LIN {X 0,Y 136.202,Z 770.659,A -85,B 0,C 180,E1 7477.588,E2 7477.588} C_VEL
LIN {X 0,Y 136.38,Z 770.694,A -85,B 0,C 180,E1 7471.676,E2 7471.676} C_VEL
LIN {X 0,Y 136.378,Z 769.624,A -85,B 0,C 180,E1 7466.633,E2 7466.633} C_VEL
LIN {X 0,Y 136.448,Z 766.979,A -85,B 0,C 180,E1 7460.718,E2 7460.718} C_VEL
LIN {X 0,Y 136.634,Z 766.026,A -85,B 0,C 180,E1 7458.6,E2 7458.6} C_VEL
LIN {X 0,Y 138.841,Z 767.204,A -85,B 0,C 180,E1 7448.274,E2 7448.274} C_VEL
LIN {X 0,Y 145.472,Z 766.561,A -85,B 0,C 180,E1 7438.042,E2 7438.042} C_VEL
LIN {X 0,Y 157.729,Z 763.951,A -85,B 0,C 180,E1 7428.267,E2 7428.267} C_VEL
LIN {X 0,Y 170.729,Z 760.685,A -85,B 0,C 180,E1 7421.759,E2 7421.759} C_VEL
LIN {X 0,Y 156.243,Z 761.337,A -85,B 0,C 180,E1 7414.272,E2 7414.272} C_VEL
LIN {X 0,Y 145.762,Z 760.293,A -85,B 0,C 180,E1 7405.603,E2 7405.603} C_VEL
LIN {X 0,Y 139.457,Z 757.48,A -85,B 0,C 180,E1 7396.236,E2 7396.236} C_VEL
LIN {X 0,Y 136.886,Z 753.335,A -85,B 0,C 180,E1 7387.553,E2 7387.553} C_VEL
LIN {X 0,Y 136.308,Z 748.658,A -85,B 0,C 180,E1 7380.419,E2 7380.419} C_VEL
LIN {X 0,Y 136.364,Z 742.798,A -85,B 0,C 180,E1 7373.684,E2 7373.684} C_VEL
LIN {X 0,Y 137.263,Z 734.901,A -85,B 0,C 180,E1 7366.519,E2 7366.519} C_VEL
LIN {X 0,Y 139.461,Z 725.036,A -85,B 0,C 180,E1 7359.431,E2 7359.431} C_VEL
LIN {X 0,Y 142.943,Z 713.689,A -85,B 0,C 180,E1 7352.955,E2 7352.955} C_VEL
LIN {X 0,Y 147.839,Z 700.038,A -85,B 0,C 180,E1 7346.781,E2 7346.781} C_VEL
LIN {X 0,Y 153.697,Z 684.691,A -85,B 0,C 180,E1 7341.325,E2 7341.325} C_VEL
LIN {X 0,Y 160.141,Z 667.742,A -85,B 0,C 180,E1 7336.621,E2 7336.621} C_VEL
LIN {X 0,Y 166.838,Z 649.18,A -85,B 0,C 180,E1 7332.63,E2 7332.63} C_VEL
LIN {X 0,Y 173.319,Z 629.638,A -85,B 0,C 180,E1 7329.371,E2 7329.371} C_VEL
LIN {X 0,Y 179.516,Z 608.54,A -85,B 0,C 180,E1 7326.672,E2 7326.672} C_VEL
LIN {X 0,Y 184.868,Z 587.205,A -85,B 0,C 180,E1 7324.607,E2 7324.607} C_VEL
LIN {X 0,Y 189.518,Z 564.355,A -85,B 0,C 180,E1 7323.014,E2 7323.014} C_VEL
LIN {X 0,Y 200.571,Z 495.538,A -85,B 0,C 180,E1 7319.493,E2 7319.493} C_VEL
LIN {X 0,Y 196.571,Z 500.049,A -85,B 0,C 180,E1 7318.892,E2 7318.892} C_VEL
LIN {X 0,Y 192.978,Z 508.1,A -85,B 0,C 180,E1 7318.713,E2 7318.713} C_VEL
LIN {X 0,Y 189.976,Z 512.133,A -85,B 0,C 180,E1 7318.319,E2 7318.319} C_VEL
LIN {X 0,Y 187.942,Z 514.262,A -85,B 0,C 180,E1 7317.832,E2 7317.832} C_VEL
LIN {X 0,Y 187.389,Z 518.122,A -85,B 0,C 180,E1 7317.404,E2 7317.404} C_VEL
LIN {X 0,Y 186.903,Z 526.414,A -85,B 0,C 180,E1 7317.05,E2 7317.05} C_VEL
LIN {X 0,Y 178.232,Z 635.184,A -85,B 0,C 180,E1 7313.3,E2 7313.3} C_VEL
LIN {X 0,Y 175.765,Z 651.989,A -85,B 0,C 180,E1 7312.165,E2 7312.165} C_VEL
LIN {X 0,Y 172.642,Z 666.742,A -85,B 0,C 180,E1 7310.692,E2 7310.692} C_VEL
LIN {X 0,Y 168.594,Z 681.234,A -85,B 0,C 180,E1 7308.682,E2 7308.682} C_VEL
LIN {X 0,Y 163.629,Z 695.775,A -85,B 0,C 180,E1 7305.964,E2 7305.964} C_VEL
LIN {X 0,Y 158.471,Z 708.511,A -85,B 0,C 180,E1 7302.762,E2 7302.762} C_VEL
LIN {X 0,Y 153.349,Z 719.856,A -85,B 0,C 180,E1 7299.007,E2 7299.007} C_VEL
LIN {X 0,Y 148.442,Z 729.85,A -85,B 0,C 180,E1 7294.64,E2 7294.64} C_VEL
LIN {X 0,Y 143.727,Z 739.095,A -85,B 0,C 180,E1 7289.207,E2 7289.207} C_VEL
LIN {X 0,Y 140.182,Z 746.209,A -85,B 0,C 180,E1 7283.452,E2 7283.452} C_VEL
LIN {X 0,Y 137.716,Z 751.82,A -85,B 0,C 180,E1 7276.998,E2 7276.998} C_VEL
LIN {X 0,Y 136.594,Z 755.376,A -85,B 0,C 180,E1 7270.773,E2 7270.773} C_VEL
LIN {X 0,Y 136.355,Z 757.366,A -85,B 0,C 180,E1 7264.371,E2 7264.371} C_VEL
LIN {X 0,Y 136.925,Z 757.835,A -85,B 0,C 180,E1 7257.793,E2 7257.793} C_VEL
LIN {X 0,Y 138.691,Z 756.654,A -85,B 0,C 180,E1 7251.135,E2 7251.135} C_VEL
LIN {X 0,Y 142.253,Z 753.429,A -85,B 0,C 180,E1 7244.205,E2 7244.205} C_VEL
LIN {X 0,Y 147.052,Z 748.647,A -85,B 0,C 180,E1 7238.226,E2 7238.226} C_VEL
LIN {X 0,Y 153.218,Z 741.888,A -85,B 0,C 180,E1 7232.676,E2 7232.676} C_VEL
LIN {X 0,Y 160.059,Z 733.612,A -85,B 0,C 180,E1 7227.939,E2 7227.939} C_VEL
LIN {X 0,Y 167.558,Z 723.336,A -85,B 0,C 180,E1 7223.747,E2 7223.747} C_VEL
LIN {X 0,Y 174.867,Z 711.855,A -85,B 0,C 180,E1 7220.34,E2 7220.34} C_VEL
LIN {X 0,Y 181.888,Z 698.953,A -85,B 0,C 180,E1 7217.509,E2 7217.509} C_VEL
LIN {X 0,Y 188.022,Z 685.344,A -85,B 0,C 180,E1 7215.305,E2 7215.305} C_VEL
LIN {X 0,Y 193.337,Z 670.636,A -85,B 0,C 180,E1 7213.545,E2 7213.545} C_VEL
LIN {X 0,Y 197.488,Z 655.424,A -85,B 0,C 180,E1 7212.23,E2 7212.23} C_VEL
LIN {X 0,Y 200.617,Z 638.603,A -85,B 0,C 180,E1 7211.246,E2 7211.246} C_VEL
LIN {X 0,Y 204.02,Z 605.103,A -85,B 0,C 180,E1 7210.152,E2 7210.152} C_VEL
LIN {X 0,Y 211.834,Z 524.075,A -85,B 0,C 180,E1 7207.779,E2 7207.779} C_VEL
LIN {X 0,Y 212.398,Z 496.448,A -85,B 0,C 180,E1 7205.573,E2 7205.573} C_VEL
LIN {X 0,Y 212.772,Z 490.461,A -85,B 0,C 180,E1 7205.02,E2 7205.02} C_VEL
LIN {X 0,Y 224.955,Z 447.879,A -85,B 0,C 180,E1 7199.89,E2 7199.89} C_VEL
LIN {X 0,Y 225.289,Z 446.689,A -85,B 0,C 180,E1 7199.747,E2 7199.747} C_VEL
LIN {X 0,Y 224.925,Z 439.714,A -85,B 0,C 180,E1 7196.433,E2 7196.433} C_VEL
LIN {X 0,Y 224.669,Z 434.477,A -85,B 0,C 180,E1 7192.917,E2 7192.917} C_VEL
LIN {X 0,Y 224.564,Z 431.171,A -85,B 0,C 180,E1 7189.714,E2 7189.714} C_VEL
LIN {X 0,Y 225.058,Z 428.722,A -85,B 0,C 180,E1 7185.858,E2 7185.858} C_VEL
LIN {X 0,Y 225.213,Z 428.615,A -85,B 0,C 180,E1 7184.024,E2 7184.024} C_VEL
LIN {X 0,Y 223.089,Z 438.023,A -85,B 0,C 180,E1 7180.503,E2 7180.503} C_VEL
LIN {X 0,Y 222.438,Z 440.67,A -85,B 0,C 180,E1 7179.938,E2 7179.938} C_VEL
LIN {X 0,Y 221.128,Z 444.689,A -85,B 0,C 180,E1 7179.659,E2 7179.659} C_VEL
LIN {X 0,Y 216.142,Z 458.259,A -85,B 0,C 180,E1 7179.808,E2 7179.808} C_VEL
LIN {X 0,Y 215.382,Z 460.548,A -85,B 0,C 180,E1 7179.71,E2 7179.71} C_VEL
LIN {X 0,Y 204.017,Z 497.28,A -85,B 0,C 180,E1 7177.4,E2 7177.4} C_VEL
LIN {X 0,Y 194.372,Z 587.356,A -85,B 0,C 180,E1 7174.197,E2 7174.197} C_VEL
LIN {X 0,Y 190.852,Z 624.419,A -85,B 0,C 180,E1 7172.598,E2 7172.598} C_VEL
LIN {X 0,Y 188.404,Z 647.642,A -85,B 0,C 180,E1 7171.449,E2 7171.449} C_VEL
LIN {X 0,Y 185.307,Z 663.835,A -85,B 0,C 180,E1 7170.239,E2 7170.239} C_VEL
LIN {X 0,Y 180.934,Z 679.336,A -85,B 0,C 180,E1 7168.617,E2 7168.617} C_VEL
LIN {X 0,Y 175.515,Z 694.069,A -85,B 0,C 180,E1 7166.563,E2 7166.563} C_VEL
LIN {X 0,Y 169.269,Z 707.769,A -85,B 0,C 180,E1 7164.015,E2 7164.015} C_VEL
LIN {X 0,Y 161.79,Z 721.666,A -85,B 0,C 180,E1 7160.572,E2 7160.572} C_VEL
LIN {X 0,Y 154.309,Z 733.62,A -85,B 0,C 180,E1 7156.522,E2 7156.522} C_VEL
LIN {X 0,Y 147.122,Z 744.014,A -85,B 0,C 180,E1 7151.754,E2 7151.754} C_VEL
LIN {X 0,Y 140.559,Z 752.753,A -85,B 0,C 180,E1 7146.181,E2 7146.181} C_VEL
LIN {X 0,Y 135.035,Z 759.962,A -85,B 0,C 180,E1 7139.736,E2 7139.736} C_VEL
LIN {X 0,Y 131.03,Z 765.309,A -85,B 0,C 180,E1 7132.586,E2 7132.586} C_VEL
LIN {X 0,Y 128.834,Z 768.723,A -85,B 0,C 180,E1 7125.294,E2 7125.294} C_VEL
LIN {X 0,Y 128.211,Z 770.292,A -85,B 0,C 180,E1 7117.951,E2 7117.951} C_VEL
LIN {X 0,Y 128.388,Z 770.241,A -85,B 0,C 180,E1 7111.78,E2 7111.78} C_VEL
LIN {X 0,Y 128.386,Z 769.096,A -85,B 0,C 180,E1 7106.423,E2 7106.423} C_VEL
LIN {X 0,Y 128.497,Z 766.359,A -85,B 0,C 180,E1 7100.138,E2 7100.138} C_VEL
LIN {X 0,Y 128.816,Z 764.854,A -85,B 0,C 180,E1 7097.443,E2 7097.443} C_VEL
LIN {X 0,Y 131.253,Z 766.254,A -85,B 0,C 180,E1 7087.134,E2 7087.134} C_VEL
LIN {X 0,Y 138.611,Z 765.981,A -85,B 0,C 180,E1 7076.255,E2 7076.255} C_VEL
LIN {X 0,Y 152.308,Z 763.787,A -85,B 0,C 180,E1 7065.899,E2 7065.899} C_VEL
LIN {X 0,Y 160.499,Z 762.17,A -85,B 0,C 180,E1 7061.711,E2 7061.711} C_VEL
LIN {X 0,Y 146.19,Z 761.822,A -85,B 0,C 180,E1 7053.64,E2 7053.64} C_VEL
LIN {X 0,Y 136.487,Z 759.886,A -85,B 0,C 180,E1 7044.679,E2 7044.679} C_VEL
LIN {X 0,Y 130.847,Z 756.352,A -85,B 0,C 180,E1 7035.057,E2 7035.057} C_VEL
LIN {X 0,Y 128.672,Z 751.44,A -85,B 0,C 180,E1 7025.796,E2 7025.796} C_VEL
LIN {X 0,Y 128.309,Z 746.391,A -85,B 0,C 180,E1 7018.659,E2 7018.659} C_VEL
LIN {X 0,Y 128.557,Z 739.855,A -85,B 0,C 180,E1 7011.5,E2 7011.5} C_VEL
LIN {X 0,Y 129.878,Z 731.149,A -85,B 0,C 180,E1 7003.908,E2 7003.908} C_VEL
LIN {X 0,Y 132.724,Z 720.359,A -85,B 0,C 180,E1 6996.466,E2 6996.466} C_VEL
LIN {X 0,Y 136.933,Z 708.027,A -85,B 0,C 180,E1 6989.745,E2 6989.745} C_VEL
LIN {X 0,Y 142.425,Z 693.704,A -85,B 0,C 180,E1 6983.613,E2 6983.613} C_VEL
LIN {X 0,Y 148.518,Z 678.345,A -85,B 0,C 180,E1 6978.459,E2 6978.459} C_VEL
LIN {X 0,Y 155.327,Z 660.805,A -85,B 0,C 180,E1 6973.864,E2 6973.864} C_VEL
LIN {X 0,Y 162.096,Z 642.235,A -85,B 0,C 180,E1 6970.102,E2 6970.102} C_VEL
LIN {X 0,Y 168.842,Z 621.674,A -85,B 0,C 180,E1 6966.92,E2 6966.92} C_VEL
LIN {X 0,Y 175.053,Z 600.001,A -85,B 0,C 180,E1 6964.374,E2 6964.374} C_VEL
LIN {X 0,Y 180.378,Z 577.861,A -85,B 0,C 180,E1 6962.439,E2 6962.439} C_VEL
LIN {X 0,Y 184.961,Z 553.44,A -85,B 0,C 180,E1 6960.942,E2 6960.942} C_VEL
LIN {X 0,Y 189.625,Z 524.883,A -85,B 0,C 180,E1 6959.422,E2 6959.422} C_VEL
LIN {X 0,Y 185.421,Z 534.382,A -85,B 0,C 180,E1 6959.255,E2 6959.255} C_VEL
LIN {X 0,Y 182.143,Z 538.992,A -85,B 0,C 180,E1 6958.845,E2 6958.845} C_VEL
LIN {X 0,Y 180.549,Z 542.085,A -85,B 0,C 180,E1 6958.47,E2 6958.47} C_VEL
LIN {X 0,Y 179.354,Z 551.32,A -85,B 0,C 180,E1 6958.045,E2 6958.045} C_VEL
LIN {X 0,Y 172.354,Z 635.636,A -85,B 0,C 180,E1 6955.07,E2 6955.07} C_VEL
LIN {X 0,Y 169.761,Z 652.518,A -85,B 0,C 180,E1 6953.913,E2 6953.913} C_VEL
LIN {X 0,Y 166.535,Z 667.111,A -85,B 0,C 180,E1 6952.433,E2 6952.433} C_VEL
LIN {X 0,Y 162.279,Z 681.697,A -85,B 0,C 180,E1 6950.376,E2 6950.376} C_VEL
LIN {X 0,Y 157.086,Z 696.228,A -85,B 0,C 180,E1 6947.602,E2 6947.602} C_VEL
LIN {X 0,Y 151.421,Z 709.519,A -85,B 0,C 180,E1 6944.146,E2 6944.146} C_VEL
LIN {X 0,Y 146.063,Z 720.768,A -85,B 0,C 180,E1 6940.256,E2 6940.256} C_VEL
LIN {X 0,Y 140.524,Z 731.368,A -85,B 0,C 180,E1 6935.312,E2 6935.312} C_VEL
LIN {X 0,Y 135.971,Z 739.819,A -85,B 0,C 180,E1 6930.005,E2 6930.005} C_VEL
LIN {X 0,Y 132.256,Z 746.841,A -85,B 0,C 180,E1 6923.929,E2 6923.929} C_VEL
LIN {X 0,Y 129.696,Z 752.395,A -85,B 0,C 180,E1 6917.086,E2 6917.086} C_VEL
LIN {X 0,Y 128.544,Z 755.948,A -85,B 0,C 180,E1 6910.256,E2 6910.256} C_VEL
LIN {X 0,Y 128.396,Z 757.896,A -85,B 0,C 180,E1 6903.155,E2 6903.155} C_VEL
LIN {X 0,Y 129.213,Z 758.215,A -85,B 0,C 180,E1 6896.148,E2 6896.148} C_VEL
LIN {X 0,Y 131.554,Z 756.704,A -85,B 0,C 180,E1 6888.804,E2 6888.804} C_VEL
LIN {X 0,Y 135.603,Z 753.414,A -85,B 0,C 180,E1 6881.873,E2 6881.873} C_VEL
LIN {X 0,Y 141.262,Z 748.146,A -85,B 0,C 180,E1 6875.481,E2 6875.481} C_VEL
LIN {X 0,Y 147.897,Z 741.367,A -85,B 0,C 180,E1 6870.02,E2 6870.02} C_VEL
LIN {X 0,Y 155.646,Z 732.426,A -85,B 0,C 180,E1 6865.084,E2 6865.084} C_VEL
LIN {X 0,Y 163.193,Z 722.607,A -85,B 0,C 180,E1 6861.193,E2 6861.193} C_VEL
LIN {X 0,Y 170.7,Z 711.251,A -85,B 0,C 180,E1 6857.926,E2 6857.926} C_VEL
LIN {X 0,Y 177.733,Z 698.817,A -85,B 0,C 180,E1 6855.265,E2 6855.265} C_VEL
LIN {X 0,Y 184.25,Z 684.766,A -85,B 0,C 180,E1 6853.06,E2 6853.06} C_VEL
LIN {X 0,Y 189.682,Z 670.139,A -85,B 0,C 180,E1 6851.368,E2 6851.368} C_VEL
LIN {X 0,Y 194.005,Z 654.43,A -85,B 0,C 180,E1 6850.073,E2 6850.073} C_VEL
LIN {X 0,Y 197.094,Z 637.969,A -85,B 0,C 180,E1 6849.154,E2 6849.154} C_VEL
LIN {X 0,Y 208.623,Z 525.21,A -85,B 0,C 180,E1 6845.796,E2 6845.796} C_VEL
LIN {X 0,Y 209.509,Z 497.097,A -85,B 0,C 180,E1 6843.507,E2 6843.507} C_VEL
LIN {X 0,Y 209.986,Z 490.835,A -85,B 0,C 180,E1 6842.913,E2 6842.913} C_VEL
LIN {X 0,Y 221.687,Z 451.523,A -85,B 0,C 180,E1 6838.224,E2 6838.224} C_VEL
LIN {X 0,Y 221.644,Z 445.832,A -85,B 0,C 180,E1 6835.343,E2 6835.343} C_VEL
LIN {X 0,Y 221.626,Z 441.035,A -85,B 0,C 180,E1 6831.961,E2 6831.961} C_VEL
LIN {X 0,Y 221.723,Z 438.353,A -85,B 0,C 180,E1 6829.083,E2 6829.083} C_VEL
LIN {X 0,Y 222.268,Z 436.205,A -85,B 0,C 180,E1 6825.676,E2 6825.676} C_VEL
LIN {X 0,Y 222.344,Z 436.178,A -85,B 0,C 180,E1 6824.615,E2 6824.615} C_VEL
LIN {X 0,Y 219.694,Z 447.341,A -85,B 0,C 180,E1 6820.491,E2 6820.491} C_VEL
LIN {X 0,Y 215.382,Z 460.548,A -85,B 0,C 180,E1 6819.71,E2 6819.71} C_VEL
LIN {X 0,Y 212.886,Z 467.853,A -85,B 0,C 180,E1 6819.514,E2 6819.514} C_VEL
LIN {X 0,Y 205.414,Z 487.684,A -85,B 0,C 180,E1 6820.021,E2 6820.021} C_VEL
LIN {X 0,Y 203.249,Z 493.872,A -85,B 0,C 180,E1 6819.814,E2 6819.814} C_VEL
LIN {X 0,Y 202.069,Z 500.702,A -85,B 0,C 180,E1 6819.5,E2 6819.5} C_VEL
LIN {X 0,Y 192.265,Z 588.417,A -85,B 0,C 180,E1 6816.467,E2 6816.467} C_VEL
LIN {X 0,Y 188.432,Z 625.593,A -85,B 0,C 180,E1 6814.875,E2 6814.875} C_VEL
LIN {X 0,Y 185.928,Z 647.063,A -85,B 0,C 180,E1 6813.826,E2 6813.826} C_VEL
LIN {X 0,Y 182.619,Z 663.38,A -85,B 0,C 180,E1 6812.656,E2 6812.656} C_VEL
LIN {X 0,Y 178.11,Z 678.587,A -85,B 0,C 180,E1 6811.124,E2 6811.124} C_VEL
LIN {X 0,Y 172.036,Z 694.227,A -85,B 0,C 180,E1 6809.002,E2 6809.002} C_VEL
LIN {X 0,Y 165.087,Z 708.426,A -85,B 0,C 180,E1 6806.377,E2 6806.377} C_VEL
LIN {X 0,Y 157.471,Z 721.539,A -85,B 0,C 180,E1 6803.126,E2 6803.126} C_VEL
LIN {X 0,Y 149.139,Z 733.82,A -85,B 0,C 180,E1 6798.929,E2 6798.929} C_VEL
LIN {X 0,Y 141.683,Z 743.714,A -85,B 0,C 180,E1 6794.311,E2 6794.311} C_VEL
LIN {X 0,Y 134.485,Z 752.399,A -85,B 0,C 180,E1 6788.64,E2 6788.64} C_VEL
LIN {X 0,Y 128.322,Z 759.579,A -85,B 0,C 180,E1 6781.989,E2 6781.989} C_VEL
LIN {X 0,Y 123.87,Z 764.727,A -85,B 0,C 180,E1 6774.812,E2 6774.812} C_VEL
LIN {X 0,Y 121.103,Z 768.31,A -85,B 0,C 180,E1 6766.791,E2 6766.791} C_VEL
LIN {X 0,Y 120.228,Z 769.872,A -85,B 0,C 180,E1 6759.086,E2 6759.086} C_VEL
LIN {X 0,Y 120.376,Z 769.844,A -85,B 0,C 180,E1 6752.375,E2 6752.375} C_VEL
LIN {X 0,Y 120.409,Z 768.863,A -85,B 0,C 180,E1 6747.139,E2 6747.139} C_VEL
LIN {X 0,Y 120.475,Z 766.241,A -85,B 0,C 180,E1 6740.44,E2 6740.44} C_VEL
LIN {X 0,Y 121.104,Z 763.691,A -85,B 0,C 180,E1 6735.654,E2 6735.654} C_VEL
LIN {X 0,Y 124.727,Z 765.297,A -85,B 0,C 180,E1 6723.833,E2 6723.833} C_VEL
LIN {X 0,Y 134.486,Z 765.11,A -85,B 0,C 180,E1 6711.892,E2 6711.892} C_VEL
LIN {X 0,Y 149.618,Z 763.223,A -85,B 0,C 180,E1 6702.111,E2 6702.111} C_VEL
LIN {X 0,Y 150.332,Z 763.087,A -85,B 0,C 180,E1 6701.688,E2 6701.688} C_VEL
LIN {X 0,Y 136.634,Z 761.817,A -85,B 0,C 180,E1 6693.285,E2 6693.285} C_VEL
LIN {X 0,Y 126.957,Z 758.851,A -85,B 0,C 180,E1 6683.188,E2 6683.188} C_VEL
LIN {X 0,Y 122.02,Z 754.358,A -85,B 0,C 180,E1 6672.78,E2 6672.78} C_VEL
LIN {X 0,Y 120.548,Z 749.125,A -85,B 0,C 180,E1 6663.803,E2 6663.803} C_VEL
LIN {X 0,Y 120.361,Z 743.74,A -85,B 0,C 180,E1 6656.665,E2 6656.665} C_VEL
LIN {X 0,Y 120.871,Z 736.504,A -85,B 0,C 180,E1 6649.03,E2 6649.03} C_VEL
LIN {X 0,Y 122.746,Z 726.938,A -85,B 0,C 180,E1 6640.982,E2 6640.982} C_VEL
LIN {X 0,Y 126.078,Z 715.923,A -85,B 0,C 180,E1 6633.632,E2 6633.632} C_VEL
LIN {X 0,Y 130.65,Z 703.573,A -85,B 0,C 180,E1 6627.085,E2 6627.085} C_VEL
LIN {X 0,Y 136.581,Z 688.898,A -85,B 0,C 180,E1 6620.979,E2 6620.979} C_VEL
LIN {X 0,Y 143.505,Z 671.986,A -85,B 0,C 180,E1 6615.553,E2 6615.553} C_VEL
LIN {X 0,Y 150.649,Z 653.881,A -85,B 0,C 180,E1 6611.081,E2 6611.081} C_VEL
LIN {X 0,Y 157.86,Z 634.093,A -85,B 0,C 180,E1 6607.352,E2 6607.352} C_VEL
LIN {X 0,Y 164.696,Z 612.92,A -85,B 0,C 180,E1 6604.343,E2 6604.343} C_VEL
LIN {X 0,Y 170.893,Z 590.458,A -85,B 0,C 180,E1 6601.963,E2 6601.963} C_VEL
LIN {X 0,Y 176.109,Z 567.407,A -85,B 0,C 180,E1 6600.197,E2 6600.197} C_VEL
LIN {X 0,Y 176.373,Z 565.822,A -85,B 0,C 180,E1 6600.091,E2 6600.091} C_VEL
LIN {X 0,Y 173.022,Z 569.857,A -85,B 0,C 180,E1 6599.518,E2 6599.518} C_VEL
LIN {X 0,Y 171.94,Z 575.214,A -85,B 0,C 180,E1 6599.172,E2 6599.172} C_VEL
LIN {X 0,Y 166.523,Z 636.559,A -85,B 0,C 180,E1 6596.913,E2 6596.913} C_VEL
LIN {X 0,Y 163.719,Z 653.78,A -85,B 0,C 180,E1 6595.701,E2 6595.701} C_VEL
LIN {X 0,Y 160.202,Z 668.669,A -85,B 0,C 180,E1 6594.133,E2 6594.133} C_VEL
LIN {X 0,Y 155.492,Z 683.807,A -85,B 0,C 180,E1 6591.902,E2 6591.902} C_VEL
LIN {X 0,Y 150.342,Z 697.358,A -85,B 0,C 180,E1 6589.195,E2 6589.195} C_VEL
LIN {X 0,Y 144.245,Z 710.887,A -85,B 0,C 180,E1 6585.522,E2 6585.522} C_VEL
LIN {X 0,Y 138.832,Z 721.611,A -85,B 0,C 180,E1 6581.624,E2 6581.624} C_VEL
LIN {X 0,Y 133.031,Z 732.092,A -85,B 0,C 180,E1 6576.478,E2 6576.478} C_VEL
LIN {X 0,Y 128.241,Z 740.48,A -85,B 0,C 180,E1 6570.898,E2 6570.898} C_VEL
LIN {X 0,Y 124.337,Z 747.428,A -85,B 0,C 180,E1 6564.468,E2 6564.468} C_VEL
LIN {X 0,Y 121.672,Z 752.937,A -85,B 0,C 180,E1 6557.186,E2 6557.186} C_VEL
LIN {X 0,Y 120.494,Z 756.527,A -85,B 0,C 180,E1 6549.609,E2 6549.609} C_VEL
LIN {X 0,Y 120.441,Z 758.339,A -85,B 0,C 180,E1 6542.303,E2 6542.303} C_VEL
LIN {X 0,Y 121.474,Z 758.594,A -85,B 0,C 180,E1 6534.825,E2 6534.825} C_VEL
LIN {X 0,Y 124.311,Z 756.97,A -85,B 0,C 180,E1 6526.876,E2 6526.876} C_VEL
LIN {X 0,Y 128.808,Z 753.656,A -85,B 0,C 180,E1 6519.791,E2 6519.791} C_VEL
LIN {X 0,Y 135.028,Z 748.367,A -85,B 0,C 180,E1 6513.212,E2 6513.212} C_VEL
LIN {X 0,Y 142.225,Z 741.57,A -85,B 0,C 180,E1 6507.646,E2 6507.646} C_VEL
LIN {X 0,Y 149.895,Z 733.32,A -85,B 0,C 180,E1 6503.011,E2 6503.011} C_VEL
LIN {X 0,Y 158.003,Z 723.418,A -85,B 0,C 180,E1 6499.025,E2 6499.025} C_VEL
LIN {X 0,Y 165.979,Z 712.006,A -85,B 0,C 180,E1 6495.73,E2 6495.73} C_VEL
LIN {X 0,Y 173.692,Z 698.979,A -85,B 0,C 180,E1 6492.975,E2 6492.975} C_VEL
LIN {X 0,Y 180.303,Z 685.283,A -85,B 0,C 180,E1 6490.869,E2 6490.869} C_VEL
LIN {X 0,Y 186.029,Z 670.575,A -85,B 0,C 180,E1 6489.195,E2 6489.195} C_VEL
LIN {X 0,Y 190.559,Z 654.845,A -85,B 0,C 180,E1 6487.92,E2 6487.92} C_VEL
LIN {X 0,Y 193.788,Z 638.429,A -85,B 0,C 180,E1 6487.022,E2 6487.022} C_VEL
LIN {X 0,Y 204.252,Z 540.88,A -85,B 0,C 180,E1 6484.199,E2 6484.199} C_VEL
LIN {X 0,Y 205.73,Z 526.209,A -85,B 0,C 180,E1 6483.739,E2 6483.739} C_VEL
LIN {X 0,Y 206.965,Z 497.506,A -85,B 0,C 180,E1 6481.357,E2 6481.357} C_VEL
LIN {X 0,Y 207.351,Z 491.943,A -85,B 0,C 180,E1 6480.83,E2 6480.83} C_VEL
LIN {X 0,Y 218.321,Z 456.356,A -85,B 0,C 180,E1 6476.621,E2 6476.621} C_VEL
LIN {X 0,Y 218.508,Z 451.219,A -85,B 0,C 180,E1 6473.696,E2 6473.696} C_VEL
LIN {X 0,Y 218.611,Z 447.258,A -85,B 0,C 180,E1 6470.524,E2 6470.524} C_VEL
LIN {X 0,Y 218.922,Z 445.339,A -85,B 0,C 180,E1 6468.141,E2 6468.141} C_VEL
LIN {X 0,Y 219.533,Z 443.702,A -85,B 0,C 180,E1 6465.258,E2 6465.258} C_VEL
LIN {X 0,Y 217.397,Z 451.382,A -85,B 0,C 180,E1 6462.388,E2 6462.388} C_VEL
LIN {X 0,Y 203.249,Z 493.872,A -85,B 0,C 180,E1 6459.814,E2 6459.814} C_VEL
LIN {X 0,Y 202.26,Z 498.075,A -85,B 0,C 180,E1 6459.759,E2 6459.759} C_VEL
LIN {X 0,Y 198.78,Z 519.875,A -85,B 0,C 180,E1 6460.87,E2 6460.87} C_VEL
LIN {X 0,Y 197.506,Z 528.802,A -85,B 0,C 180,E1 6460.868,E2 6460.868} C_VEL
LIN {X 0,Y 190.628,Z 588.142,A -85,B 0,C 180,E1 6458.825,E2 6458.825} C_VEL
LIN {X 0,Y 186.453,Z 626.377,A -85,B 0,C 180,E1 6457.237,E2 6457.237} C_VEL
LIN {X 0,Y 183.974,Z 646.407,A -85,B 0,C 180,E1 6456.275,E2 6456.275} C_VEL
LIN {X 0,Y 180.416,Z 662.83,A -85,B 0,C 180,E1 6455.151,E2 6455.151} C_VEL
LIN {X 0,Y 175.31,Z 678.869,A -85,B 0,C 180,E1 6453.587,E2 6453.587} C_VEL
LIN {X 0,Y 168.886,Z 694.356,A -85,B 0,C 180,E1 6451.533,E2 6451.533} C_VEL
LIN {X 0,Y 161.203,Z 709.08,A -85,B 0,C 180,E1 6448.855,E2 6448.855} C_VEL
LIN {X 0,Y 153.5,Z 721.472,A -85,B 0,C 180,E1 6445.808,E2 6445.808} C_VEL
LIN {X 0,Y 144.943,Z 733.227,A -85,B 0,C 180,E1 6441.843,E2 6441.843} C_VEL
LIN {X 0,Y 136.559,Z 743.443,A -85,B 0,C 180,E1 6437.062,E2 6437.062} C_VEL
LIN {X 0,Y 128.697,Z 752.084,A -85,B 0,C 180,E1 6431.321,E2 6431.321} C_VEL
LIN {X 0,Y 121.835,Z 759.211,A -85,B 0,C 180,E1 6424.483,E2 6424.483} C_VEL
LIN {X 0,Y 116.493,Z 764.602,A -85,B 0,C 180,E1 6416.501,E2 6416.501} C_VEL
LIN {X 0,Y 113.45,Z 767.902,A -85,B 0,C 180,E1 6408.492,E2 6408.492} C_VEL
LIN {X 0,Y 112.268,Z 769.46,A -85,B 0,C 180,E1 6400.255,E2 6400.255} C_VEL
LIN {X 0,Y 112.358,Z 769.441,A -85,B 0,C 180,E1 6393.055,E2 6393.055} C_VEL
LIN {X 0,Y 112.427,Z 768.471,A -85,B 0,C 180,E1 6387.446,E2 6387.446} C_VEL
LIN {X 0,Y 112.49,Z 765.856,A -85,B 0,C 180,E1 6380.272,E2 6380.272} C_VEL
LIN {X 0,Y 113.523,Z 762.407,A -85,B 0,C 180,E1 6373.624,E2 6373.624} C_VEL
LIN {X 0,Y 118.347,Z 764.275,A -85,B 0,C 180,E1 6360.653,E2 6360.653} C_VEL
LIN {X 0,Y 129.663,Z 764.361,A -85,B 0,C 180,E1 6348.453,E2 6348.453} C_VEL
LIN {X 0,Y 140.208,Z 763.444,A -85,B 0,C 180,E1 6341.68,E2 6341.68} C_VEL
LIN {X 0,Y 126.639,Z 761.21,A -85,B 0,C 180,E1 6332.47,E2 6332.47} C_VEL
LIN {X 0,Y 117.821,Z 757.452,A -85,B 0,C 180,E1 6321.923,E2 6321.923} C_VEL
LIN {X 0,Y 113.602,Z 752.346,A -85,B 0,C 180,E1 6311.163,E2 6311.163} C_VEL
LIN {X 0,Y 112.526,Z 746.75,A -85,B 0,C 180,E1 6302.035,E2 6302.035} C_VEL
LIN {X 0,Y 112.485,Z 740.692,A -85,B 0,C 180,E1 6294.387,E2 6294.387} C_VEL
LIN {X 0,Y 113.448,Z 732.262,A -85,B 0,C 180,E1 6285.826,E2 6285.826} C_VEL
LIN {X 0,Y 115.92,Z 722.215,A -85,B 0,C 180,E1 6277.694,E2 6277.694} C_VEL
LIN {X 0,Y 120.065,Z 710.209,A -85,B 0,C 180,E1 6270.014,E2 6270.014} C_VEL
LIN {X 0,Y 125.684,Z 696.284,A -85,B 0,C 180,E1 6263.083,E2 6263.083} C_VEL
LIN {X 0,Y 132.27,Z 680.786,A -85,B 0,C 180,E1 6257.128,E2 6257.128} C_VEL
LIN {X 0,Y 139.729,Z 663.027,A -85,B 0,C 180,E1 6251.908,E2 6251.908} C_VEL
LIN {X 0,Y 147.2,Z 644.11,A -85,B 0,C 180,E1 6247.69,E2 6247.69} C_VEL
LIN {X 0,Y 154.363,Z 624.096,A -85,B 0,C 180,E1 6244.305,E2 6244.305} C_VEL
LIN {X 0,Y 161.807,Z 603.088,A -85,B 0,C 180,E1 6241.273,E2 6241.273} C_VEL
LIN {X 0,Y 164.493,Z 598.733,A -85,B 0,C 180,E1 6240.38,E2 6240.38} C_VEL
LIN {X 0,Y 160.873,Z 637.386,A -85,B 0,C 180,E1 6238.888,E2 6238.888} C_VEL
LIN {X 0,Y 157.89,Z 654.784,A -85,B 0,C 180,E1 6237.641,E2 6237.641} C_VEL
LIN {X 0,Y 154.053,Z 670.031,A -85,B 0,C 180,E1 6235.987,E2 6235.987} C_VEL
LIN {X 0,Y 149.146,Z 684.985,A -85,B 0,C 180,E1 6233.722,E2 6233.722} C_VEL
LIN {X 0,Y 143.783,Z 698.304,A -85,B 0,C 180,E1 6230.97,E2 6230.97} C_VEL
LIN {X 0,Y 137.405,Z 711.746,A -85,B 0,C 180,E1 6227.199,E2 6227.199} C_VEL
LIN {X 0,Y 131.214,Z 723.232,A -85,B 0,C 180,E1 6222.771,E2 6222.771} C_VEL
LIN {X 0,Y 125.17,Z 733.536,A -85,B 0,C 180,E1 6217.348,E2 6217.348} C_VEL
LIN {X 0,Y 120.012,Z 741.969,A -85,B 0,C 180,E1 6211.163,E2 6211.163} C_VEL
LIN {X 0,Y 115.964,Z 748.873,A -85,B 0,C 180,E1 6204.067,E2 6204.067} C_VEL
LIN {X 0,Y 113.521,Z 753.745,A -85,B 0,C 180,E1 6196.768,E2 6196.768} C_VEL
LIN {X 0,Y 112.436,Z 757.188,A -85,B 0,C 180,E1 6188.623,E2 6188.623} C_VEL
LIN {X 0,Y 112.552,Z 758.865,A -85,B 0,C 180,E1 6180.758,E2 6180.758} C_VEL
LIN {X 0,Y 113.957,Z 758.904,A -85,B 0,C 180,E1 6172.749,E2 6172.749} C_VEL
LIN {X 0,Y 117.476,Z 757.108,A -85,B 0,C 180,E1 6164.263,E2 6164.263} C_VEL
LIN {X 0,Y 122.637,Z 753.604,A -85,B 0,C 180,E1 6156.975,E2 6156.975} C_VEL
LIN {X 0,Y 129.62,Z 748.167,A -85,B 0,C 180,E1 6150.249,E2 6150.249} C_VEL
LIN {X 0,Y 137.503,Z 741.119,A -85,B 0,C 180,E1 6144.653,E2 6144.653} C_VEL
LIN {X 0,Y 145.8,Z 732.663,A -85,B 0,C 180,E1 6140.045,E2 6140.045} C_VEL
LIN {X 0,Y 154.332,Z 722.595,A -85,B 0,C 180,E1 6136.177,E2 6136.177} C_VEL
LIN {X 0,Y 163.058,Z 710.546,A -85,B 0,C 180,E1 6132.866,E2 6132.866} C_VEL
LIN {X 0,Y 170.737,Z 697.845,A -85,B 0,C 180,E1 6130.342,E2 6130.342} C_VEL
LIN {X 0,Y 177.81,Z 683.535,A -85,B 0,C 180,E1 6128.269,E2 6128.269} C_VEL
LIN {X 0,Y 183.475,Z 668.875,A -85,B 0,C 180,E1 6126.729,E2 6126.729} C_VEL
LIN {X 0,Y 188.147,Z 652.528,A -85,B 0,C 180,E1 6125.509,E2 6125.509} C_VEL
LIN {X 0,Y 191.133,Z 636.436,A -85,B 0,C 180,E1 6124.722,E2 6124.722} C_VEL
LIN {X 0,Y 203.102,Z 527.428,A -85,B 0,C 180,E1 6121.641,E2 6121.641} C_VEL
LIN {X 0,Y 204.787,Z 498.053,A -85,B 0,C 180,E1 6119.162,E2 6119.162} C_VEL
LIN {X 0,Y 205.236,Z 492.312,A -85,B 0,C 180,E1 6118.605,E2 6118.605} C_VEL
LIN {X 0,Y 215.194,Z 461.424,A -85,B 0,C 180,E1 6115.003,E2 6115.003} C_VEL
LIN {X 0,Y 215.522,Z 456.686,A -85,B 0,C 180,E1 6112.001,E2 6112.001} C_VEL
LIN {X 0,Y 216.015,Z 453.147,A -85,B 0,C 180,E1 6108.521,E2 6108.521} C_VEL
LIN {X 0,Y 216.573,Z 451.528,A -85,B 0,C 180,E1 6105.801,E2 6105.801} C_VEL
LIN {X 0,Y 215.212,Z 455.651,A -85,B 0,C 180,E1 6104.299,E2 6104.299} C_VEL
LIN {X 0,Y 201.415,Z 496.274,A -85,B 0,C 180,E1 6101.939,E2 6101.939} C_VEL
LIN {X 0,Y 197.506,Z 528.802,A -85,B 0,C 180,E1 6100.868,E2 6100.868} C_VEL
LIN {X 0,Y 196.46,Z 536.496,A -85,B 0,C 180,E1 6100.911,E2 6100.911} C_VEL
LIN {X 0,Y 193.175,Z 557.118,A -85,B 0,C 180,E1 6102.035,E2 6102.035} C_VEL
LIN {X 0,Y 192.278,Z 563.71,A -85,B 0,C 180,E1 6102.034,E2 6102.034} C_VEL
LIN {X 0,Y 188.845,Z 591.771,A -85,B 0,C 180,E1 6101.101,E2 6101.101} C_VEL
LIN {X 0,Y 183.238,Z 640.154,A -85,B 0,C 180,E1 6099.072,E2 6099.072} C_VEL
LIN {X 0,Y 180.226,Z 656.172,A -85,B 0,C 180,E1 6098.133,E2 6098.133} C_VEL
LIN {X 0,Y 176.001,Z 670.839,A -85,B 0,C 180,E1 6096.962,E2 6096.962} C_VEL
LIN {X 0,Y 170.343,Z 685.58,A -85,B 0,C 180,E1 6095.372,E2 6095.372} C_VEL
LIN {X 0,Y 163.383,Z 699.895,A -85,B 0,C 180,E1 6093.304,E2 6093.304} C_VEL
LIN {X 0,Y 154.654,Z 714.434,A -85,B 0,C 180,E1 6090.398,E2 6090.398} C_VEL
LIN {X 0,Y 146.309,Z 726.212,A -85,B 0,C 180,E1 6087.191,E2 6087.191} C_VEL
LIN {X 0,Y 136.813,Z 737.724,A -85,B 0,C 180,E1 6082.798,E2 6082.798} C_VEL
LIN {X 0,Y 128.198,Z 746.932,A -85,B 0,C 180,E1 6077.803,E2 6077.803} C_VEL
LIN {X 0,Y 119.51,Z 755.281,A -85,B 0,C 180,E1 6071.154,E2 6071.154} C_VEL
LIN {X 0,Y 112.825,Z 761.327,A -85,B 0,C 180,E1 6063.932,E2 6063.932} C_VEL
LIN {X 0,Y 107.686,Z 765.854,A -85,B 0,C 180,E1 6055.277,E2 6055.277} C_VEL
LIN {X 0,Y 104.977,Z 768.395,A -85,B 0,C 180,E1 6046.596,E2 6046.596} C_VEL
LIN {X 0,Y 104.235,Z 769.208,A -85,B 0,C 180,E1 6037.712,E2 6037.712} C_VEL
LIN {X 0,Y 104.471,Z 768.618,A -85,B 0,C 180,E1 6030.542,E2 6030.542} C_VEL
LIN {X 0,Y 104.396,Z 766.96,A -85,B 0,C 180,E1 6023.947,E2 6023.947} C_VEL
LIN {X 0,Y 105.046,Z 763.277,A -85,B 0,C 180,E1 6015.666,E2 6015.666} C_VEL
LIN {X 0,Y 106.049,Z 760.985,A -85,B 0,C 180,E1 6011.582,E2 6011.582} C_VEL
LIN {X 0,Y 111.495,Z 763.024,A -85,B 0,C 180,E1 5998.419,E2 5998.419} C_VEL
LIN {X 0,Y 124.247,Z 763.462,A -85,B 0,C 180,E1 5985.557,E2 5985.557} C_VEL
LIN {X 0,Y 130.103,Z 763.244,A -85,B 0,C 180,E1 5981.662,E2 5981.662} C_VEL
LIN {X 0,Y 116.705,Z 760.043,A -85,B 0,C 180,E1 5971.506,E2 5971.506} C_VEL
LIN {X 0,Y 108.529,Z 755.342,A -85,B 0,C 180,E1 5959.928,E2 5959.928} C_VEL
LIN {X 0,Y 105.183,Z 749.524,A -85,B 0,C 180,E1 5948.621,E2 5948.621} C_VEL
LIN {X 0,Y 104.542,Z 743.958,A -85,B 0,C 180,E1 5939.998,E2 5939.998} C_VEL
LIN {X 0,Y 104.707,Z 737.221,A -85,B 0,C 180,E1 5931.763,E2 5931.763} C_VEL
LIN {X 0,Y 106.104,Z 728.423,A -85,B 0,C 180,E1 5923.013,E2 5923.013} C_VEL
LIN {X 0,Y 109.224,Z 717.705,A -85,B 0,C 180,E1 5914.515,E2 5914.515} C_VEL
LIN {X 0,Y 113.812,Z 705.683,A -85,B 0,C 180,E1 5906.995,E2 5906.995} C_VEL
LIN {X 0,Y 120.178,Z 690.866,A -85,B 0,C 180,E1 5899.848,E2 5899.848} C_VEL
LIN {X 0,Y 127.482,Z 674.351,A -85,B 0,C 180,E1 5893.813,E2 5893.813} C_VEL
LIN {X 0,Y 135.883,Z 655.591,A -85,B 0,C 180,E1 5888.401,E2 5888.401} C_VEL
LIN {X 0,Y 137.445,Z 653.713,A -85,B 0,C 180,E1 5887.537,E2 5887.537} C_VEL
LIN {X 0,Y 141.396,Z 650.325,A -85,B 0,C 180,E1 5885.934,E2 5885.934} C_VEL
LIN {X 0,Y 147.121,Z 643.313,A -85,B 0,C 180,E1 5884.161,E2 5884.161} C_VEL
LIN {X 0,Y 153.534,Z 632.723,A -85,B 0,C 180,E1 5882.416,E2 5882.416} C_VEL
LIN {X 0,Y 156.742,Z 626.402,A -85,B 0,C 180,E1 5881.543,E2 5881.543} C_VEL
LIN {X 0,Y 154.573,Z 643.891,A -85,B 0,C 180,E1 5880.663,E2 5880.663} C_VEL
LIN {X 0,Y 151.036,Z 660.847,A -85,B 0,C 180,E1 5879.228,E2 5879.228} C_VEL
LIN {X 0,Y 146.743,Z 675.625,A -85,B 0,C 180,E1 5877.413,E2 5877.413} C_VEL
LIN {X 0,Y 140.968,Z 691.1,A -85,B 0,C 180,E1 5874.743,E2 5874.743} C_VEL
LIN {X 0,Y 134.859,Z 704.513,A -85,B 0,C 180,E1 5871.535,E2 5871.535} C_VEL
LIN {X 0,Y 128.291,Z 716.957,A -85,B 0,C 180,E1 5867.466,E2 5867.466} C_VEL
LIN {X 0,Y 121.953,Z 727.637,A -85,B 0,C 180,E1 5862.663,E2 5862.663} C_VEL
LIN {X 0,Y 115.623,Z 737.575,A -85,B 0,C 180,E1 5856.46,E2 5856.46} C_VEL
LIN {X 0,Y 110.526,Z 745.408,A -85,B 0,C 180,E1 5849.487,E2 5849.487} C_VEL
LIN {X 0,Y 106.76,Z 751.735,A -85,B 0,C 180,E1 5841.388,E2 5841.388} C_VEL
LIN {X 0,Y 104.797,Z 756.066,A -85,B 0,C 180,E1 5832.803,E2 5832.803} C_VEL
LIN {X 0,Y 104.379,Z 758.599,A -85,B 0,C 180,E1 5824.221,E2 5824.221} C_VEL
LIN {X 0,Y 105.213,Z 759.499,A -85,B 0,C 180,E1 5815.773,E2 5815.773} C_VEL
LIN {X 0,Y 107.995,Z 758.675,A -85,B 0,C 180,E1 5806.764,E2 5806.764} C_VEL
LIN {X 0,Y 112.72,Z 756.181,A -85,B 0,C 180,E1 5798.696,E2 5798.696} C_VEL
LIN {X 0,Y 119.467,Z 751.721,A -85,B 0,C 180,E1 5791.26,E2 5791.26} C_VEL
LIN {X 0,Y 127.342,Z 745.736,A -85,B 0,C 180,E1 5785.089,E2 5785.089} C_VEL
LIN {X 0,Y 136.408,Z 737.692,A -85,B 0,C 180,E1 5779.707,E2 5779.707} C_VEL
LIN {X 0,Y 145.802,Z 728.085,A -85,B 0,C 180,E1 5775.313,E2 5775.313} C_VEL
LIN {X 0,Y 154.519,Z 717.547,A -85,B 0,C 180,E1 5771.952,E2 5771.952} C_VEL
LIN {X 0,Y 163.036,Z 705.406,A -85,B 0,C 180,E1 5769.145,E2 5769.145} C_VEL
LIN {X 0,Y 170.624,Z 692.227,A -85,B 0,C 180,E1 5766.945,E2 5766.945} C_VEL
LIN {X 0,Y 177.363,Z 677.73,A -85,B 0,C 180,E1 5765.176,E2 5765.176} C_VEL
LIN {X 0,Y 182.738,Z 662.521,A -85,B 0,C 180,E1 5763.843,E2 5763.843} C_VEL
LIN {X 0,Y 186.878,Z 646.156,A -85,B 0,C 180,E1 5762.846,E2 5762.846} C_VEL
LIN {X 0,Y 189.47,Z 628.853,A -85,B 0,C 180,E1 5762.187,E2 5762.187} C_VEL
LIN {X 0,Y 200.875,Z 528.69,A -85,B 0,C 180,E1 5759.484,E2 5759.484} C_VEL
LIN {X 0,Y 202.968,Z 498.374,A -85,B 0,C 180,E1 5756.895,E2 5756.895} C_VEL
LIN {X 0,Y 203.464,Z 492.715,A -85,B 0,C 180,E1 5756.338,E2 5756.338} C_VEL
LIN {X 0,Y 212.252,Z 466.698,A -85,B 0,C 180,E1 5753.374,E2 5753.374} C_VEL
LIN {X 0,Y 212.753,Z 462.41,A -85,B 0,C 180,E1 5750.26,E2 5750.26} C_VEL
LIN {X 0,Y 213.323,Z 460.166,A -85,B 0,C 180,E1 5747.55,E2 5747.55} C_VEL
LIN {X 0,Y 213.55,Z 459.604,A -85,B 0,C 180,E1 5746.281,E2 5746.281} C_VEL
LIN {X 0,Y 206.277,Z 479.499,A -85,B 0,C 180,E1 5745.227,E2 5745.227} C_VEL
LIN {X 0,Y 200.62,Z 496.182,A -85,B 0,C 180,E1 5744.246,E2 5744.246} C_VEL
LIN {X 0,Y 196.225,Z 531.683,A -85,B 0,C 180,E1 5743.101,E2 5743.101} C_VEL
LIN {X 0,Y 192.278,Z 563.71,A -85,B 0,C 180,E1 5742.034,E2 5742.034} C_VEL
LIN {X 0,Y 191.218,Z 571.41,A -85,B 0,C 180,E1 5742.081,E2 5742.081} C_VEL
LIN {X 0,Y 188.027,Z 592.044,A -85,B 0,C 180,E1 5743.307,E2 5743.307} C_VEL
LIN {X 0,Y 187.137,Z 598.641,A -85,B 0,C 180,E1 5743.303,E2 5743.303} C_VEL
LIN {X 0,Y 181.549,Z 642.927,A -85,B 0,C 180,E1 5741.421,E2 5741.421} C_VEL
LIN {X 0,Y 178.106,Z 658.435,A -85,B 0,C 180,E1 5740.51,E2 5740.51} C_VEL
LIN {X 0,Y 173.62,Z 672.664,A -85,B 0,C 180,E1 5739.395,E2 5739.395} C_VEL
LIN {X 0,Y 167.783,Z 686.835,A -85,B 0,C 180,E1 5737.909,E2 5737.909} C_VEL
LIN {X 0,Y 160.423,Z 700.898,A -85,B 0,C 180,E1 5735.923,E2 5735.923} C_VEL
LIN {X 0,Y 151.679,Z 714.614,A -85,B 0,C 180,E1 5733.268,E2 5733.268} C_VEL
LIN {X 0,Y 142.874,Z 726.156,A -85,B 0,C 180,E1 5730.191,E2 5730.191} C_VEL
LIN {X 0,Y 132.777,Z 737.57,A -85,B 0,C 180,E1 5725.919,E2 5725.919} C_VEL
LIN {X 0,Y 123.517,Z 746.711,A -85,B 0,C 180,E1 5720.988,E2 5720.988} C_VEL
LIN {X 0,Y 114.193,Z 754.872,A -85,B 0,C 180,E1 5714.456,E2 5714.456} C_VEL
LIN {X 0,Y 106.548,Z 760.985,A -85,B 0,C 180,E1 5706.904,E2 5706.904} C_VEL
LIN {X 0,Y 100.347,Z 765.697,A -85,B 0,C 180,E1 5697.273,E2 5697.273} C_VEL
LIN {X 0,Y 97.203,Z 768.077,A -85,B 0,C 180,E1 5687.967,E2 5687.967} C_VEL
LIN {X 0,Y 96.247,Z 768.788,A -85,B 0,C 180,E1 5678.356,E2 5678.356} C_VEL
LIN {X 0,Y 96.485,Z 768.103,A -85,B 0,C 180,E1 5670.587,E2 5670.587} C_VEL
LIN {X 0,Y 96.408,Z 766.344,A -85,B 0,C 180,E1 5663.443,E2 5663.443} C_VEL
LIN {X 0,Y 97.352,Z 762.248,A -85,B 0,C 180,E1 5653.894,E2 5653.894} C_VEL
LIN {X 0,Y 98.808,Z 759.526,A -85,B 0,C 180,E1 5648.94,E2 5648.94} C_VEL
LIN {X 0,Y 106.5,Z 761.861,A -85,B 0,C 180,E1 5633.732,E2 5633.732} C_VEL
LIN {X 0,Y 120.177,Z 762.512,A -85,B 0,C 180,E1 5621.726,E2 5621.726} C_VEL
LIN {X 0,Y 106.854,Z 758.318,A -85,B 0,C 180,E1 5610.349,E2 5610.349} C_VEL
LIN {X 0,Y 99.417,Z 752.664,A -85,B 0,C 180,E1 5597.559,E2 5597.559} C_VEL
LIN {X 0,Y 96.969,Z 746.324,A -85,B 0,C 180,E1 5585.916,E2 5585.916} C_VEL
LIN {X 0,Y 96.615,Z 740.733,A -85,B 0,C 180,E1 5577.625,E2 5577.625} C_VEL
LIN {X 0,Y 97.166,Z 732.736,A -85,B 0,C 180,E1 5568.121,E2 5568.121} C_VEL
LIN {X 0,Y 99.565,Z 722.256,A -85,B 0,C 180,E1 5558.186,E2 5558.186} C_VEL
LIN {X 0,Y 103.846,Z 710.271,A -85,B 0,C 180,E1 5549.314,E2 5549.314} C_VEL
LIN {X 0,Y 110.06,Z 695.883,A -85,B 0,C 180,E1 5541.18,E2 5541.18} C_VEL
LIN {X 0,Y 118.936,Z 677.163,A -85,B 0,C 180,E1 5533.171,E2 5533.171} C_VEL
LIN {X 0,Y 120.78,Z 675.735,A -85,B 0,C 180,E1 5531.834,E2 5531.834} C_VEL
LIN {X 0,Y 124.934,Z 673.109,A -85,B 0,C 180,E1 5529.796,E2 5529.796} C_VEL
LIN {X 0,Y 130.437,Z 668.144,A -85,B 0,C 180,E1 5527.854,E2 5527.854} C_VEL
LIN {X 0,Y 137.482,Z 660.57,A -85,B 0,C 180,E1 5525.813,E2 5525.813} C_VEL
LIN {X 0,Y 142.414,Z 656.825,A -85,B 0,C 180,E1 5524.057,E2 5524.057} C_VEL
LIN {X 0,Y 148.096,Z 650.898,A -85,B 0,C 180,E1 5522.461,E2 5522.461} C_VEL
LIN {X 0,Y 144.107,Z 666.795,A -85,B 0,C 180,E1 5520.897,E2 5520.897} C_VEL
LIN {X 0,Y 139.079,Z 681.818,A -85,B 0,C 180,E1 5518.799,E2 5518.799} C_VEL
LIN {X 0,Y 132.823,Z 696.614,A -85,B 0,C 180,E1 5515.893,E2 5515.893} C_VEL
LIN {X 0,Y 126.221,Z 709.615,A -85,B 0,C 180,E1 5512.353,E2 5512.353} C_VEL
LIN {X 0,Y 118.94,Z 722.063,A -85,B 0,C 180,E1 5507.621,E2 5507.621} C_VEL
LIN {X 0,Y 112.445,Z 732.001,A -85,B 0,C 180,E1 5502.328,E2 5502.328} C_VEL
LIN {X 0,Y 106.079,Z 741.221,A -85,B 0,C 180,E1 5495.414,E2 5495.414} C_VEL
LIN {X 0,Y 101.226,Z 748.293,A -85,B 0,C 180,E1 5487.742,E2 5487.742} C_VEL
LIN {X 0,Y 97.873,Z 753.921,A -85,B 0,C 180,E1 5478.744,E2 5478.744} C_VEL
LIN {X 0,Y 96.521,Z 757.407,A -85,B 0,C 180,E1 5470.018,E2 5470.018} C_VEL
LIN {X 0,Y 96.537,Z 759.397,A -85,B 0,C 180,E1 5460.878,E2 5460.878} C_VEL
LIN {X 0,Y 98.131,Z 759.858,A -85,B 0,C 180,E1 5451.581,E2 5451.581} C_VEL
LIN {X 0,Y 101.812,Z 758.65,A -85,B 0,C 180,E1 5442.572,E2 5442.572} C_VEL
LIN {X 0,Y 108.18,Z 755.398,A -85,B 0,C 180,E1 5433.682,E2 5433.682} C_VEL
LIN {X 0,Y 116.08,Z 750.436,A -85,B 0,C 180,E1 5426.401,E2 5426.401} C_VEL
LIN {X 0,Y 125.614,Z 743.4,A -85,B 0,C 180,E1 5420.09,E2 5420.09} C_VEL
LIN {X 0,Y 134.821,Z 735.39,A -85,B 0,C 180,E1 5415.419,E2 5415.419} C_VEL
LIN {X 0,Y 144.8,Z 725.195,A -85,B 0,C 180,E1 5411.352,E2 5411.352} C_VEL
LIN {X 0,Y 153.602,Z 714.534,A -85,B 0,C 180,E1 5408.37,E2 5408.37} C_VEL
LIN {X 0,Y 162.092,Z 702.21,A -85,B 0,C 180,E1 5405.879,E2 5405.879} C_VEL
LIN {X 0,Y 169.85,Z 688.529,A -85,B 0,C 180,E1 5403.871,E2 5403.871} C_VEL
LIN {X 0,Y 176.597,Z 673.419,A -85,B 0,C 180,E1 5402.273,E2 5402.273} C_VEL
LIN {X 0,Y 181.755,Z 658.082,A -85,B 0,C 180,E1 5401.112,E2 5401.112} C_VEL
LIN {X 0,Y 185.599,Z 641.233,A -85,B 0,C 180,E1 5400.249,E2 5400.249} C_VEL
LIN {X 0,Y 189.124,Z 613.558,A -85,B 0,C 180,E1 5399.429,E2 5399.429} C_VEL
LIN {X 0,Y 198.993,Z 529.77,A -85,B 0,C 180,E1 5397.265,E2 5397.265} C_VEL
LIN {X 0,Y 201.501,Z 499.378,A -85,B 0,C 180,E1 5394.645,E2 5394.645} C_VEL
LIN {X 0,Y 202.492,Z 492.06,A -85,B 0,C 180,E1 5393.907,E2 5393.907} C_VEL
LIN {X 0,Y 209.424,Z 472.054,A -85,B 0,C 180,E1 5391.628,E2 5391.628} C_VEL
LIN {X 0,Y 210.157,Z 468.73,A -85,B 0,C 180,E1 5388.752,E2 5388.752} C_VEL
LIN {X 0,Y 210.313,Z 468.219,A -85,B 0,C 180,E1 5387.988,E2 5387.988} C_VEL
LIN {X 0,Y 200.315,Z 495.616,A -85,B 0,C 180,E1 5386.605,E2 5386.605} C_VEL
LIN {X 0,Y 197.502,Z 517.258,A -85,B 0,C 180,E1 5385.846,E2 5385.846} C_VEL
LIN {X 0,Y 188.07,Z 591.227,A -85,B 0,C 180,E1 5383.546,E2 5383.546} C_VEL
LIN {X 0,Y 187.137,Z 598.641,A -85,B 0,C 180,E1 5383.303,E2 5383.303} C_VEL
LIN {X 0,Y 186.104,Z 606.325,A -85,B 0,C 180,E1 5383.307,E2 5383.307} C_VEL
LIN {X 0,Y 183.049,Z 627.011,A -85,B 0,C 180,E1 5384.399,E2 5384.399} C_VEL
LIN {X 0,Y 182.139,Z 633.602,A -85,B 0,C 180,E1 5384.395,E2 5384.395} C_VEL
LIN {X 0,Y 179.13,Z 650.536,A -85,B 0,C 180,E1 5383.595,E2 5383.595} C_VEL
LIN {X 0,Y 174.484,Z 666.732,A -85,B 0,C 180,E1 5382.56,E2 5382.56} C_VEL
LIN {X 0,Y 168.449,Z 681.944,A -85,B 0,C 180,E1 5381.202,E2 5381.202} C_VEL
LIN {X 0,Y 160.342,Z 697.689,A -85,B 0,C 180,E1 5379.274,E2 5379.274} C_VEL
LIN {X 0,Y 151.57,Z 711.36,A -85,B 0,C 180,E1 5376.948,E2 5376.948} C_VEL
LIN {X 0,Y 141.459,Z 724.416,A -85,B 0,C 180,E1 5373.841,E2 5373.841} C_VEL
LIN {X 0,Y 131.424,Z 735.267,A -85,B 0,C 180,E1 5370.135,E2 5370.135} C_VEL
LIN {X 0,Y 121.323,Z 744.716,A -85,B 0,C 180,E1 5365.49,E2 5365.49} C_VEL
LIN {X 0,Y 111.521,Z 752.787,A -85,B 0,C 180,E1 5359.639,E2 5359.639} C_VEL
LIN {X 0,Y 102.063,Z 759.683,A -85,B 0,C 180,E1 5351.763,E2 5351.763} C_VEL
LIN {X 0,Y 95.159,Z 764.255,A -85,B 0,C 180,E1 5343.11,E2 5343.11} C_VEL
LIN {X 0,Y 90.167,Z 767.357,A -85,B 0,C 180,E1 5332.142,E2 5332.142} C_VEL
LIN {X 0,Y 88.358,Z 768.391,A -85,B 0,C 180,E1 5321.745,E2 5321.745} C_VEL
LIN {X 0,Y 88.417,Z 767.892,A -85,B 0,C 180,E1 5312.586,E2 5312.586} C_VEL
LIN {X 0,Y 88.438,Z 766.638,A -85,B 0,C 180,E1 5306.103,E2 5306.103} C_VEL
LIN {X 0,Y 88.885,Z 763.346,A -85,B 0,C 180,E1 5296.329,E2 5296.329} C_VEL
LIN {X 0,Y 91.828,Z 757.904,A -85,B 0,C 180,E1 5285.894,E2 5285.894} C_VEL
LIN {X 0,Y 101.042,Z 760.514,A -85,B 0,C 180,E1 5269.961,E2 5269.961} C_VEL
LIN {X 0,Y 110.236,Z 761.227,A -85,B 0,C 180,E1 5261.742,E2 5261.742} C_VEL
LIN {X 0,Y 97.038,Z 755.99,A -85,B 0,C 180,E1 5248.845,E2 5248.845} C_VEL
LIN {X 0,Y 90.694,Z 749.71,A -85,B 0,C 180,E1 5235.34,E2 5235.34} C_VEL
LIN {X 0,Y 88.962,Z 743.307,A -85,B 0,C 180,E1 5223.864,E2 5223.864} C_VEL
LIN {X 0,Y 88.758,Z 737.547,A -85,B 0,C 180,E1 5215.475,E2 5215.475} C_VEL
LIN {X 0,Y 89.716,Z 728.861,A -85,B 0,C 180,E1 5205.145,E2 5205.145} C_VEL
LIN {X 0,Y 92.715,Z 718.079,A -85,B 0,C 180,E1 5194.956,E2 5194.956} C_VEL
LIN {X 0,Y 97.747,Z 705.492,A -85,B 0,C 180,E1 5185.762,E2 5185.762} C_VEL
LIN {X 0,Y 103.832,Z 692.715,A -85,B 0,C 180,E1 5178.357,E2 5178.357} C_VEL
LIN {X 0,Y 105.291,Z 691.668,A -85,B 0,C 180,E1 5176.862,E2 5176.862} C_VEL
LIN {X 0,Y 109.019,Z 689.73,A -85,B 0,C 180,E1 5174.324,E2 5174.324} C_VEL
LIN {X 0,Y 115.039,Z 685.431,A -85,B 0,C 180,E1 5171.626,E2 5171.626} C_VEL
LIN {X 0,Y 118.258,Z 682.828,A -85,B 0,C 180,E1 5170.45,E2 5170.45} C_VEL
LIN {X 0,Y 122.432,Z 680.806,A -85,B 0,C 180,E1 5168.369,E2 5168.369} C_VEL
LIN {X 0,Y 128.761,Z 676.171,A -85,B 0,C 180,E1 5166.136,E2 5166.136} C_VEL
LIN {X 0,Y 138.249,Z 666.859,A -85,B 0,C 180,E1 5163.722,E2 5163.722} C_VEL
LIN {X 0,Y 139.018,Z 666.57,A -85,B 0,C 180,E1 5163.402,E2 5163.402} C_VEL
LIN {X 0,Y 133.704,Z 681.929,A -85,B 0,C 180,E1 5161.289,E2 5161.289} C_VEL
LIN {X 0,Y 127.234,Z 696.614,A -85,B 0,C 180,E1 5158.418,E2 5158.418} C_VEL
LIN {X 0,Y 120.594,Z 709.195,A -85,B 0,C 180,E1 5155.02,E2 5155.02} C_VEL
LIN {X 0,Y 112.859,Z 721.778,A -85,B 0,C 180,E1 5150.219,E2 5150.219} C_VEL
LIN {X 0,Y 105.907,Z 731.877,A -85,B 0,C 180,E1 5144.774,E2 5144.774} C_VEL
LIN {X 0,Y 99.024,Z 741.193,A -85,B 0,C 180,E1 5137.549,E2 5137.549} C_VEL
LIN {X 0,Y 93.722,Z 748.386,A -85,B 0,C 180,E1 5129.395,E2 5129.395} C_VEL
LIN {X 0,Y 90.043,Z 754.054,A -85,B 0,C 180,E1 5119.773,E2 5119.773} C_VEL
LIN {X 0,Y 88.531,Z 757.68,A -85,B 0,C 180,E1 5110.203,E2 5110.203} C_VEL
LIN {X 0,Y 88.573,Z 759.725,A -85,B 0,C 180,E1 5100.373,E2 5100.373} C_VEL
LIN {X 0,Y 90.6,Z 760.265,A -85,B 0,C 180,E1 5089.598,E2 5089.598} C_VEL
LIN {X 0,Y 94.993,Z 759,A -85,B 0,C 180,E1 5079.803,E2 5079.803} C_VEL
LIN {X 0,Y 102.174,Z 755.748,A -85,B 0,C 180,E1 5070.567,E2 5070.567} C_VEL
LIN {X 0,Y 110.419,Z 751.058,A -85,B 0,C 180,E1 5063.482,E2 5063.482} C_VEL
LIN {X 0,Y 120.399,Z 744.251,A -85,B 0,C 180,E1 5057.269,E2 5057.269} C_VEL
LIN {X 0,Y 130.125,Z 736.406,A -85,B 0,C 180,E1 5052.643,E2 5052.643} C_VEL
LIN {X 0,Y 140.571,Z 726.341,A -85,B 0,C 180,E1 5048.662,E2 5048.662} C_VEL
LIN {X 0,Y 150.194,Z 715.369,A -85,B 0,C 180,E1 5045.644,E2 5045.644} C_VEL
LIN {X 0,Y 159.215,Z 702.911,A -85,B 0,C 180,E1 5043.214,E2 5043.214} C_VEL
LIN {X 0,Y 167.011,Z 689.834,A -85,B 0,C 180,E1 5041.366,E2 5041.366} C_VEL
LIN {X 0,Y 173.615,Z 675.831,A -85,B 0,C 180,E1 5039.923,E2 5039.923} C_VEL
LIN {X 0,Y 179,Z 660.951,A -85,B 0,C 180,E1 5038.807,E2 5038.807} C_VEL
LIN {X 0,Y 183.01,Z 645.247,A -85,B 0,C 180,E1 5037.986,E2 5037.986} C_VEL
LIN {X 0,Y 185.876,Z 626.11,A -85,B 0,C 180,E1 5037.365,E2 5037.365} C_VEL
LIN {X 0,Y 197.404,Z 530.969,A -85,B 0,C 180,E1 5035.016,E2 5035.016} C_VEL
LIN {X 0,Y 200.381,Z 500.425,A -85,B 0,C 180,E1 5032.367,E2 5032.367} C_VEL
LIN {X 0,Y 201.509,Z 492.591,A -85,B 0,C 180,E1 5031.584,E2 5031.584} C_VEL
LIN {X 0,Y 206.852,Z 477.796,A -85,B 0,C 180,E1 5029.98,E2 5029.98} C_VEL
LIN {X 0,Y 206.855,Z 477.728,A -85,B 0,C 180,E1 5029.796,E2 5029.796} C_VEL
LIN {X 0,Y 200.331,Z 495.442,A -85,B 0,C 180,E1 5028.946,E2 5028.946} C_VEL
LIN {X 0,Y 198.215,Z 510.88,A -85,B 0,C 180,E1 5028.346,E2 5028.346} C_VEL
LIN {X 0,Y 189.294,Z 578.105,A -85,B 0,C 180,E1 5026.327,E2 5026.327} C_VEL
LIN {X 0,Y 185.604,Z 606.428,A -85,B 0,C 180,E1 5025.447,E2 5025.447} C_VEL
LIN {X 0,Y 182.139,Z 633.602,A -85,B 0,C 180,E1 5024.395,E2 5024.395} C_VEL
LIN {X 0,Y 180.92,Z 641.274,A -85,B 0,C 180,E1 5024.46,E2 5024.46} C_VEL
LIN {X 0,Y 176.871,Z 657.395,A -85,B 0,C 180,E1 5025.261,E2 5025.261} C_VEL
LIN {X 0,Y 174.09,Z 665.779,A -85,B 0,C 180,E1 5025.253,E2 5025.253} C_VEL
LIN {X 0,Y 173.374,Z 667.819,A -85,B 0,C 180,E1 5025.145,E2 5025.145} C_VEL
LIN {X 0,Y 166.583,Z 683.75,A -85,B 0,C 180,E1 5023.795,E2 5023.795} C_VEL
LIN {X 0,Y 158.64,Z 698.254,A -85,B 0,C 180,E1 5022.105,E2 5022.105} C_VEL
LIN {X 0,Y 149.523,Z 711.588,A -85,B 0,C 180,E1 5019.957,E2 5019.957} C_VEL
LIN {X 0,Y 138.97,Z 724.496,A -85,B 0,C 180,E1 5017.049,E2 5017.049} C_VEL
LIN {X 0,Y 128.415,Z 735.25,A -85,B 0,C 180,E1 5013.548,E2 5013.548} C_VEL
LIN {X 0,Y 117.666,Z 744.635,A -85,B 0,C 180,E1 5009.108,E2 5009.108} C_VEL
LIN {X 0,Y 107.08,Z 752.555,A -85,B 0,C 180,E1 5003.409,E2 5003.409} C_VEL
LIN {X 0,Y 96.662,Z 759.388,A -85,B 0,C 180,E1 4995.529,E2 4995.529} C_VEL
LIN {X 0,Y 88.83,Z 763.907,A -85,B 0,C 180,E1 4986.615,E2 4986.615} C_VEL
LIN {X 0,Y 82.896,Z 766.977,A -85,B 0,C 180,E1 4974.962,E2 4974.962} C_VEL
LIN {X 0,Y 80.502,Z 767.97,A -85,B 0,C 180,E1 4963.642,E2 4963.642} C_VEL
LIN {X 0,Y 80.39,Z 767.466,A -85,B 0,C 180,E1 4953.558,E2 4953.558} C_VEL
LIN {X 0,Y 80.473,Z 766.373,A -85,B 0,C 180,E1 4947.144,E2 4947.144} C_VEL
LIN {X 0,Y 80.766,Z 763.426,A -85,B 0,C 180,E1 4937.117,E2 4937.117} C_VEL
LIN {X 0,Y 83.246,Z 758.568,A -85,B 0,C 180,E1 4926.642,E2 4926.642} C_VEL
LIN {X 0,Y 85.166,Z 756.173,A -85,B 0,C 180,E1 4922.364,E2 4922.364} C_VEL
LIN {X 0,Y 96.108,Z 758.934,A -85,B 0,C 180,E1 4905.802,E2 4905.802} C_VEL
LIN {X 0,Y 100.46,Z 759.439,A -85,B 0,C 180,E1 4901.821,E2 4901.821} C_VEL
LIN {X 0,Y 87.854,Z 753.433,A -85,B 0,C 180,E1 4887.813,E2 4887.813} C_VEL
LIN {X 0,Y 82.289,Z 746.59,A -85,B 0,C 180,E1 4873.345,E2 4873.345} C_VEL
LIN {X 0,Y 81.03,Z 740.337,A -85,B 0,C 180,E1 4862.119,E2 4862.119} C_VEL
LIN {X 0,Y 81.014,Z 733.468,A -85,B 0,C 180,E1 4852.195,E2 4852.195} C_VEL
LIN {X 0,Y 82.679,Z 723.905,A -85,B 0,C 180,E1 4840.94,E2 4840.94} C_VEL
LIN {X 0,Y 86.675,Z 712.325,A -85,B 0,C 180,E1 4830.259,E2 4830.259} C_VEL
LIN {X 0,Y 89.909,Z 705.194,A -85,B 0,C 180,E1 4824.667,E2 4824.667} C_VEL
LIN {X 0,Y 93.73,Z 703.212,A -85,B 0,C 180,E1 4820.202,E2 4820.202} C_VEL
LIN {X 0,Y 99.145,Z 700.001,A -85,B 0,C 180,E1 4816.701,E2 4816.701} C_VEL
LIN {X 0,Y 101.986,Z 698.217,A -85,B 0,C 180,E1 4815.097,E2 4815.097} C_VEL
LIN {X 0,Y 106.526,Z 696.253,A -85,B 0,C 180,E1 4812.137,E2 4812.137} C_VEL
LIN {X 0,Y 112.676,Z 692.477,A -85,B 0,C 180,E1 4809.461,E2 4809.461} C_VEL
LIN {X 0,Y 117.65,Z 688.952,A -85,B 0,C 180,E1 4807.777,E2 4807.777} C_VEL
LIN {X 0,Y 122.934,Z 686.293,A -85,B 0,C 180,E1 4805.574,E2 4805.574} C_VEL
LIN {X 0,Y 128.274,Z 682.808,A -85,B 0,C 180,E1 4803.853,E2 4803.853} C_VEL
LIN {X 0,Y 121.466,Z 697.509,A -85,B 0,C 180,E1 4800.968,E2 4800.968} C_VEL
LIN {X 0,Y 114.185,Z 710.484,A -85,B 0,C 180,E1 4797.374,E2 4797.374} C_VEL
LIN {X 0,Y 106.384,Z 722.448,A -85,B 0,C 180,E1 4792.671,E2 4792.671} C_VEL
LIN {X 0,Y 99.006,Z 732.483,A -85,B 0,C 180,E1 4787.036,E2 4787.036} C_VEL
LIN {X 0,Y 91.654,Z 741.765,A -85,B 0,C 180,E1 4779.425,E2 4779.425} C_VEL
LIN {X 0,Y 85.964,Z 748.909,A -85,B 0,C 180,E1 4770.674,E2 4770.674} C_VEL
LIN {X 0,Y 82.037,Z 754.55,A -85,B 0,C 180,E1 4760.183,E2 4760.183} C_VEL
LIN {X 0,Y 80.493,Z 758.137,A -85,B 0,C 180,E1 4749.655,E2 4749.655} C_VEL
LIN {X 0,Y 80.643,Z 760.087,A -85,B 0,C 180,E1 4739.456,E2 4739.456} C_VEL
LIN {X 0,Y 83.067,Z 760.678,A -85,B 0,C 180,E1 4727.63,E2 4727.63} C_VEL
LIN {X 0,Y 88.241,Z 759.445,A -85,B 0,C 180,E1 4716.912,E2 4716.912} C_VEL
LIN {X 0,Y 96.441,Z 756.144,A -85,B 0,C 180,E1 4707.143,E2 4707.143} C_VEL
LIN {X 0,Y 105.534,Z 751.404,A -85,B 0,C 180,E1 4699.944,E2 4699.944} C_VEL
LIN {X 0,Y 116.327,Z 744.542,A -85,B 0,C 180,E1 4693.795,E2 4693.795} C_VEL
LIN {X 0,Y 126.642,Z 736.699,A -85,B 0,C 180,E1 4689.321,E2 4689.321} C_VEL
LIN {X 0,Y 137.608,Z 726.695,A -85,B 0,C 180,E1 4685.53,E2 4685.53} C_VEL
LIN {X 0,Y 147.467,Z 715.938,A -85,B 0,C 180,E1 4682.722,E2 4682.722} C_VEL
LIN {X 0,Y 157.117,Z 703.061,A -85,B 0,C 180,E1 4680.366,E2 4680.366} C_VEL
LIN {X 0,Y 165.295,Z 689.668,A -85,B 0,C 180,E1 4678.615,E2 4678.615} C_VEL
LIN {X 0,Y 172.16,Z 675.328,A -85,B 0,C 180,E1 4677.258,E2 4677.258} C_VEL
LIN {X 0,Y 177.62,Z 660.411,A -85,B 0,C 180,E1 4676.234,E2 4676.234} C_VEL
LIN {X 0,Y 181.652,Z 644.499,A -85,B 0,C 180,E1 4675.477,E2 4675.477} C_VEL
LIN {X 0,Y 184.606,Z 624.815,A -85,B 0,C 180,E1 4674.894,E2 4674.894} C_VEL
LIN {X 0,Y 196.284,Z 532.135,A -85,B 0,C 180,E1 4672.725,E2 4672.725} C_VEL
LIN {X 0,Y 198.811,Z 508.879,A -85,B 0,C 180,E1 4670.726,E2 4670.726} C_VEL
LIN {X 0,Y 188.945,Z 580.191,A -85,B 0,C 180,E1 4668.695,E2 4668.695} C_VEL
LIN {X 0,Y 185.287,Z 607.063,A -85,B 0,C 180,E1 4667.914,E2 4667.914} C_VEL
LIN {X 0,Y 180.198,Z 643.184,A -85,B 0,C 180,E1 4666.525,E2 4666.525} C_VEL
LIN {X 0,Y 176.075,Z 659.703,A -85,B 0,C 180,E1 4665.658,E2 4665.658} C_VEL
LIN {X 0,Y 173.374,Z 667.819,A -85,B 0,C 180,E1 4665.145,E2 4665.145} C_VEL
LIN {X 0,Y 170.527,Z 675.034,A -85,B 0,C 180,E1 4664.948,E2 4664.948} C_VEL
LIN {X 0,Y 162.894,Z 689.902,A -85,B 0,C 180,E1 4665.326,E2 4665.326} C_VEL
LIN {X 0,Y 158.251,Z 697.43,A -85,B 0,C 180,E1 4665.122,E2 4665.122} C_VEL
LIN {X 0,Y 157.069,Z 699.222,A -85,B 0,C 180,E1 4664.94,E2 4664.94} C_VEL
LIN {X 0,Y 147.018,Z 713.143,A -85,B 0,C 180,E1 4662.832,E2 4662.832} C_VEL
LIN {X 0,Y 136.938,Z 724.638,A -85,B 0,C 180,E1 4660.357,E2 4660.357} C_VEL
LIN {X 0,Y 125.676,Z 735.412,A -85,B 0,C 180,E1 4657.057,E2 4657.057} C_VEL
LIN {X 0,Y 114.499,Z 744.553,A -85,B 0,C 180,E1 4652.95,E2 4652.95} C_VEL
LIN {X 0,Y 103.147,Z 752.381,A -85,B 0,C 180,E1 4647.482,E2 4647.482} C_VEL
LIN {X 0,Y 91.726,Z 759.126,A -85,B 0,C 180,E1 4639.721,E2 4639.721} C_VEL
LIN {X 0,Y 82.399,Z 763.775,A -85,B 0,C 180,E1 4630.014,E2 4630.014} C_VEL
LIN {X 0,Y 75.86,Z 766.598,A -85,B 0,C 180,E1 4618.317,E2 4618.317} C_VEL
LIN {X 0,Y 72.641,Z 767.542,A -85,B 0,C 180,E1 4605.151,E2 4605.151} C_VEL
LIN {X 0,Y 72.425,Z 766.832,A -85,B 0,C 180,E1 4593.157,E2 4593.157} C_VEL
LIN {X 0,Y 72.478,Z 765.784,A -85,B 0,C 180,E1 4586.828,E2 4586.828} C_VEL
LIN {X 0,Y 72.915,Z 762.719,A -85,B 0,C 180,E1 4575.702,E2 4575.702} C_VEL
LIN {X 0,Y 75.889,Z 757.673,A -85,B 0,C 180,E1 4564.22,E2 4564.22} C_VEL
LIN {X 0,Y 78.9,Z 754.318,A -85,B 0,C 180,E1 4558.262,E2 4558.262} C_VEL
LIN {X 0,Y 90.825,Z 757.158,A -85,B 0,C 180,E1 4541.948,E2 4541.948} C_VEL
LIN {X 0,Y 78.705,Z 750.338,A -85,B 0,C 180,E1 4526.397,E2 4526.397} C_VEL
LIN {X 0,Y 74.013,Z 743.023,A -85,B 0,C 180,E1 4510.899,E2 4510.899} C_VEL
LIN {X 0,Y 73.132,Z 736.982,A -85,B 0,C 180,E1 4499.997,E2 4499.997} C_VEL
LIN {X 0,Y 73.439,Z 729.182,A -85,B 0,C 180,E1 4488.639,E2 4488.639} C_VEL
LIN {X 0,Y 75.876,Z 719.073,A -85,B 0,C 180,E1 4476.711,E2 4476.711} C_VEL
LIN {X 0,Y 77.262,Z 715.627,A -85,B 0,C 180,E1 4472.648,E2 4472.648} C_VEL
LIN {X 0,Y 80.016,Z 714.206,A -85,B 0,C 180,E1 4467.496,E2 4467.496} C_VEL
LIN {X 0,Y 85.277,Z 711.198,A -85,B 0,C 180,E1 4462.43,E2 4462.43} C_VEL
LIN {X 0,Y 87.014,Z 710.408,A -85,B 0,C 180,E1 4460.8,E2 4460.8} C_VEL
LIN {X 0,Y 91.723,Z 708.571,A -85,B 0,C 180,E1 4456.623,E2 4456.623} C_VEL
LIN {X 0,Y 99.196,Z 704.36,A -85,B 0,C 180,E1 4452.621,E2 4452.621} C_VEL
LIN {X 0,Y 104.742,Z 702.123,A -85,B 0,C 180,E1 4449.353,E2 4449.353} C_VEL
LIN {X 0,Y 112.023,Z 698.059,A -85,B 0,C 180,E1 4446.551,E2 4446.551} C_VEL
LIN {X 0,Y 117.176,Z 694.798,A -85,B 0,C 180,E1 4444.996,E2 4444.996} C_VEL
LIN {X 0,Y 117.963,Z 694.596,A -85,B 0,C 180,E1 4444.609,E2 4444.609} C_VEL
LIN {X 0,Y 109.975,Z 708.678,A -85,B 0,C 180,E1 4441.008,E2 4441.008} C_VEL
LIN {X 0,Y 102.217,Z 720.24,A -85,B 0,C 180,E1 4436.748,E2 4436.748} C_VEL
LIN {X 0,Y 93.527,Z 731.572,A -85,B 0,C 180,E1 4430.665,E2 4430.665} C_VEL
LIN {X 0,Y 85.954,Z 740.513,A -85,B 0,C 180,E1 4423.46,E2 4423.46} C_VEL
LIN {X 0,Y 79.179,Z 748.334,A -85,B 0,C 180,E1 4413.935,E2 4413.935} C_VEL
LIN {X 0,Y 74.669,Z 754.044,A -85,B 0,C 180,E1 4403.087,E2 4403.087} C_VEL
LIN {X 0,Y 72.552,Z 758.154,A -85,B 0,C 180,E1 4390.695,E2 4390.695} C_VEL
LIN {X 0,Y 72.636,Z 760.318,A -85,B 0,C 180,E1 4379.392,E2 4379.392} C_VEL
LIN {X 0,Y 75.016,Z 761.116,A -85,B 0,C 180,E1 4367.149,E2 4367.149} C_VEL
LIN {X 0,Y 80.68,Z 760.183,A -85,B 0,C 180,E1 4355.137,E2 4355.137} C_VEL
LIN {X 0,Y 88.875,Z 757.43,A -85,B 0,C 180,E1 4345.312,E2 4345.312} C_VEL
LIN {X 0,Y 99.392,Z 752.664,A -85,B 0,C 180,E1 4337.146,E2 4337.146} C_VEL
LIN {X 0,Y 110.101,Z 746.582,A -85,B 0,C 180,E1 4331.284,E2 4331.284} C_VEL
LIN {X 0,Y 121.751,Z 738.511,A -85,B 0,C 180,E1 4326.492,E2 4326.492} C_VEL
LIN {X 0,Y 132.424,Z 729.588,A -85,B 0,C 180,E1 4323.031,E2 4323.031} C_VEL
LIN {X 0,Y 143.517,Z 718.31,A -85,B 0,C 180,E1 4320.084,E2 4320.084} C_VEL
LIN {X 0,Y 153.065,Z 706.554,A -85,B 0,C 180,E1 4317.937,E2 4317.937} C_VEL
LIN {X 0,Y 162.337,Z 692.374,A -85,B 0,C 180,E1 4316.113,E2 4316.113} C_VEL
LIN {X 0,Y 169.658,Z 678.327,A -85,B 0,C 180,E1 4314.812,E2 4314.812} C_VEL
LIN {X 0,Y 175.677,Z 663.027,A -85,B 0,C 180,E1 4313.793,E2 4313.793} C_VEL
LIN {X 0,Y 180.127,Z 647.184,A -85,B 0,C 180,E1 4313.054,E2 4313.054} C_VEL
LIN {X 0,Y 183.131,Z 629.093,A -85,B 0,C 180,E1 4312.515,E2 4312.515} C_VEL
LIN {X 0,Y 190.142,Z 574.634,A -85,B 0,C 180,E1 4311.312,E2 4311.312} C_VEL
LIN {X 0,Y 185.241,Z 609.39,A -85,B 0,C 180,E1 4310.311,E2 4310.311} C_VEL
LIN {X 0,Y 180.208,Z 642.95,A -85,B 0,C 180,E1 4309.109,E2 4309.109} C_VEL
LIN {X 0,Y 175.745,Z 659.909,A -85,B 0,C 180,E1 4308.291,E2 4308.291} C_VEL
LIN {X 0,Y 170.109,Z 674.932,A -85,B 0,C 180,E1 4307.324,E2 4307.324} C_VEL
LIN {X 0,Y 162.33,Z 690.556,A -85,B 0,C 180,E1 4305.937,E2 4305.937} C_VEL
LIN {X 0,Y 157.069,Z 699.222,A -85,B 0,C 180,E1 4304.94,E2 4304.94} C_VEL
LIN {X 0,Y 152.613,Z 705.585,A -85,B 0,C 180,E1 4304.474,E2 4304.474} C_VEL
LIN {X 0,Y 141.802,Z 718.379,A -85,B 0,C 180,E1 4304.343,E2 4304.343} C_VEL
LIN {X 0,Y 135.709,Z 724.556,A -85,B 0,C 180,E1 4303.782,E2 4303.782} C_VEL
LIN {X 0,Y 134.225,Z 725.992,A -85,B 0,C 180,E1 4303.487,E2 4303.487} C_VEL
LIN {X 0,Y 122.691,Z 736.321,A -85,B 0,C 180,E1 4300.482,E2 4300.482} C_VEL
LIN {X 0,Y 110.223,Z 745.581,A -85,B 0,C 180,E1 4296.36,E2 4296.36} C_VEL
LIN {X 0,Y 97.48,Z 753.566,A -85,B 0,C 180,E1 4290.66,E2 4290.66} C_VEL
LIN {X 0,Y 85.991,Z 759.5,A -85,B 0,C 180,E1 4283.337,E2 4283.337} C_VEL
LIN {X 0,Y 75.778,Z 763.884,A -85,B 0,C 180,E1 4273.312,E2 4273.312} C_VEL
LIN {X 0,Y 68.438,Z 766.402,A -85,B 0,C 180,E1 4260.742,E2 4260.742} C_VEL
LIN {X 0,Y 64.726,Z 767.11,A -85,B 0,C 180,E1 4246.134,E2 4246.134} C_VEL
LIN {X 0,Y 64.428,Z 766.293,A -85,B 0,C 180,E1 4233.549,E2 4233.549} C_VEL
LIN {X 0,Y 64.482,Z 765.187,A -85,B 0,C 180,E1 4226.434,E2 4226.434} C_VEL
LIN {X 0,Y 65.116,Z 761.97,A -85,B 0,C 180,E1 4213.945,E2 4213.945} C_VEL
LIN {X 0,Y 69.056,Z 756.343,A -85,B 0,C 180,E1 4200.499,E2 4200.499} C_VEL
LIN {X 0,Y 73.135,Z 752.298,A -85,B 0,C 180,E1 4193.498,E2 4193.498} C_VEL
LIN {X 0,Y 81.293,Z 754.38,A -85,B 0,C 180,E1 4182.089,E2 4182.089} C_VEL
LIN {X 0,Y 69.996,Z 747.071,A -85,B 0,C 180,E1 4165.371,E2 4165.371} C_VEL
LIN {X 0,Y 66.064,Z 739.825,A -85,B 0,C 180,E1 4149.58,E2 4149.58} C_VEL
LIN {X 0,Y 65.329,Z 734.226,A -85,B 0,C 180,E1 4139.12,E2 4139.12} C_VEL
LIN {X 0,Y 65.969,Z 725.345,A -85,B 0,C 180,E1 4125.065,E2 4125.065} C_VEL
LIN {X 0,Y 68.122,Z 723.565,A -85,B 0,C 180,E1 4116.65,E2 4116.65} C_VEL
LIN {X 0,Y 72.331,Z 721.023,A -85,B 0,C 180,E1 4110.152,E2 4110.152} C_VEL
LIN {X 0,Y 75.822,Z 719.697,A -85,B 0,C 180,E1 4104.53,E2 4104.53} C_VEL
LIN {X 0,Y 82.187,Z 716.544,A -85,B 0,C 180,E1 4098.929,E2 4098.929} C_VEL
LIN {X 0,Y 89.21,Z 713.971,A -85,B 0,C 180,E1 4093.234,E2 4093.234} C_VEL
LIN {X 0,Y 97.089,Z 710.026,A -85,B 0,C 180,E1 4089.428,E2 4089.428} C_VEL
LIN {X 0,Y 103.855,Z 707.383,A -85,B 0,C 180,E1 4086.027,E2 4086.027} C_VEL
LIN {X 0,Y 106.393,Z 706.31,A -85,B 0,C 180,E1 4084.985,E2 4084.985} C_VEL
LIN {X 0,Y 97.549,Z 719.192,A -85,B 0,C 180,E1 4080.568,E2 4080.568} C_VEL
LIN {X 0,Y 89.15,Z 729.674,A -85,B 0,C 180,E1 4075.233,E2 4075.233} C_VEL
LIN {X 0,Y 80.731,Z 739.119,A -85,B 0,C 180,E1 4068.045,E2 4068.045} C_VEL
LIN {X 0,Y 73.695,Z 746.58,A -85,B 0,C 180,E1 4059.379,E2 4059.379} C_VEL
LIN {X 0,Y 67.814,Z 753.089,A -85,B 0,C 180,E1 4047.474,E2 4047.474} C_VEL
LIN {X 0,Y 64.921,Z 757.44,A -85,B 0,C 180,E1 4034.832,E2 4034.832} C_VEL
LIN {X 0,Y 64.45,Z 760.077,A -85,B 0,C 180,E1 4022.171,E2 4022.171} C_VEL
LIN {X 0,Y 66.412,Z 761.418,A -85,B 0,C 180,E1 4008.528,E2 4008.528} C_VEL
LIN {X 0,Y 71.987,Z 761.119,A -85,B 0,C 180,E1 3994.984,E2 3994.984} C_VEL
LIN {X 0,Y 80.809,Z 758.834,A -85,B 0,C 180,E1 3983.728,E2 3983.728} C_VEL
LIN {X 0,Y 91.592,Z 754.786,A -85,B 0,C 180,E1 3975.191,E2 3975.191} C_VEL
LIN {X 0,Y 103.211,Z 749.027,A -85,B 0,C 180,E1 3968.881,E2 3968.881} C_VEL
LIN {X 0,Y 115.589,Z 741.414,A -85,B 0,C 180,E1 3963.97,E2 3963.97} C_VEL
LIN {X 0,Y 127.033,Z 732.691,A -85,B 0,C 180,E1 3960.453,E2 3960.453} C_VEL
LIN {X 0,Y 139.102,Z 721.545,A -85,B 0,C 180,E1 3957.481,E2 3957.481} C_VEL
LIN {X 0,Y 149.898,Z 709.196,A -85,B 0,C 180,E1 3955.267,E2 3955.267} C_VEL
LIN {X 0,Y 158.934,Z 696.532,A -85,B 0,C 180,E1 3953.668,E2 3953.668} C_VEL
LIN {X 0,Y 167.103,Z 682.021,A -85,B 0,C 180,E1 3952.355,E2 3952.355} C_VEL
LIN {X 0,Y 173.545,Z 667.21,A -85,B 0,C 180,E1 3951.386,E2 3951.386} C_VEL
LIN {X 0,Y 176.21,Z 659.357,A -85,B 0,C 180,E1 3950.966,E2 3950.966} C_VEL
LIN {X 0,Y 170.487,Z 674.177,A -85,B 0,C 180,E1 3950.128,E2 3950.128} C_VEL
LIN {X 0,Y 162.496,Z 689.733,A -85,B 0,C 180,E1 3948.915,E2 3948.915} C_VEL
LIN {X 0,Y 153.174,Z 704.064,A -85,B 0,C 180,E1 3947.367,E2 3947.367} C_VEL
LIN {X 0,Y 142.145,Z 717.745,A -85,B 0,C 180,E1 3945.261,E2 3945.261} C_VEL
LIN {X 0,Y 134.225,Z 725.992,A -85,B 0,C 180,E1 3943.487,E2 3943.487} C_VEL
LIN {X 0,Y 128.623,Z 731.089,A -85,B 0,C 180,E1 3942.633,E2 3942.633} C_VEL
LIN {X 0,Y 116.138,Z 740.451,A -85,B 0,C 180,E1 3941.82,E2 3941.82} C_VEL
LIN {X 0,Y 108.922,Z 745.09,A -85,B 0,C 180,E1 3940.76,E2 3940.76} C_VEL
LIN {X 0,Y 106.387,Z 746.674,A -85,B 0,C 180,E1 3940.031,E2 3940.031} C_VEL
LIN {X 0,Y 93.756,Z 753.811,A -85,B 0,C 180,E1 3935.006,E2 3935.006} C_VEL
LIN {X 0,Y 80.647,Z 759.857,A -85,B 0,C 180,E1 3927.45,E2 3927.45} C_VEL
LIN {X 0,Y 69.454,Z 763.951,A -85,B 0,C 180,E1 3917.225,E2 3917.225} C_VEL
LIN {X 0,Y 60.793,Z 766.268,A -85,B 0,C 180,E1 3902.858,E2 3902.858} C_VEL
LIN {X 0,Y 56.725,Z 766.625,A -85,B 0,C 180,E1 3886.369,E2 3886.369} C_VEL
LIN {X 0,Y 56.508,Z 765.497,A -85,B 0,C 180,E1 3872.017,E2 3872.017} C_VEL
LIN {X 0,Y 56.474,Z 763.867,A -85,B 0,C 180,E1 3862.485,E2 3862.485} C_VEL
LIN {X 0,Y 58.195,Z 759.958,A -85,B 0,C 180,E1 3847.78,E2 3847.78} C_VEL
LIN {X 0,Y 63.488,Z 754.1,A -85,B 0,C 180,E1 3834.347,E2 3834.347} C_VEL
LIN {X 0,Y 68.116,Z 750.143,A -85,B 0,C 180,E1 3827.801,E2 3827.801} C_VEL
LIN {X 0,Y 71.993,Z 751.186,A -85,B 0,C 180,E1 3822.394,E2 3822.394} C_VEL
LIN {X 0,Y 61.378,Z 743.366,A -85,B 0,C 180,E1 3804.029,E2 3804.029} C_VEL
LIN {X 0,Y 58.154,Z 736.312,A -85,B 0,C 180,E1 3787.902,E2 3787.902} C_VEL
LIN {X 0,Y 57.519,Z 734.41,A -85,B 0,C 180,E1 3781.989,E2 3781.989} C_VEL
LIN {X 0,Y 58.411,Z 731.695,A -85,B 0,C 180,E1 3768.143,E2 3768.143} C_VEL
LIN {X 0,Y 60.125,Z 730.132,A -85,B 0,C 180,E1 3762.579,E2 3762.579} C_VEL
LIN {X 0,Y 62.947,Z 728.562,A -85,B 0,C 180,E1 3753.588,E2 3753.588} C_VEL
LIN {X 0,Y 67.604,Z 726.252,A -85,B 0,C 180,E1 3746.819,E2 3746.819} C_VEL
LIN {X 0,Y 72.235,Z 724.628,A -85,B 0,C 180,E1 3740.448,E2 3740.448} C_VEL
LIN {X 0,Y 79.823,Z 721.449,A -85,B 0,C 180,E1 3734.436,E2 3734.436} C_VEL
LIN {X 0,Y 86.103,Z 719.412,A -85,B 0,C 180,E1 3729.963,E2 3729.963} C_VEL
LIN {X 0,Y 95.461,Z 715.31,A -85,B 0,C 180,E1 3725.795,E2 3725.795} C_VEL
LIN {X 0,Y 85.963,Z 727.021,A -85,B 0,C 180,E1 3720.598,E2 3720.598} C_VEL
LIN {X 0,Y 76.762,Z 736.948,A -85,B 0,C 180,E1 3713.824,E2 3713.824} C_VEL
LIN {X 0,Y 68.066,Z 745.467,A -85,B 0,C 180,E1 3704.47,E2 3704.47} C_VEL
LIN {X 0,Y 61.42,Z 752.029,A -85,B 0,C 180,E1 3692.809,E2 3692.809} C_VEL
LIN {X 0,Y 57.272,Z 757.066,A -85,B 0,C 180,E1 3677.881,E2 3677.881} C_VEL
LIN {X 0,Y 56.402,Z 759.99,A -85,B 0,C 180,E1 3663.705,E2 3663.705} C_VEL
LIN {X 0,Y 58.328,Z 761.709,A -85,B 0,C 180,E1 3648.061,E2 3648.061} C_VEL
LIN {X 0,Y 64.301,Z 761.713,A -85,B 0,C 180,E1 3632.913,E2 3632.913} C_VEL
LIN {X 0,Y 73.795,Z 759.875,A -85,B 0,C 180,E1 3620.816,E2 3620.816} C_VEL
LIN {X 0,Y 85.758,Z 755.977,A -85,B 0,C 180,E1 3611.701,E2 3611.701} C_VEL
LIN {X 0,Y 97.46,Z 750.884,A -85,B 0,C 180,E1 3605.723,E2 3605.723} C_VEL
LIN {X 0,Y 110.023,Z 743.873,A -85,B 0,C 180,E1 3601.043,E2 3601.043} C_VEL
LIN {X 0,Y 122.076,Z 735.631,A -85,B 0,C 180,E1 3597.614,E2 3597.614} C_VEL
LIN {X 0,Y 133.472,Z 726.12,A -85,B 0,C 180,E1 3595.022,E2 3595.022} C_VEL
LIN {X 0,Y 145.103,Z 714.153,A -85,B 0,C 180,E1 3592.825,E2 3592.825} C_VEL
LIN {X 0,Y 154.758,Z 701.944,A -85,B 0,C 180,E1 3591.271,E2 3591.271} C_VEL
LIN {X 0,Y 156.744,Z 699.029,A -85,B 0,C 180,E1 3590.946,E2 3590.946} C_VEL
LIN {X 0,Y 146.94,Z 711.745,A -85,B 0,C 180,E1 3589.474,E2 3589.474} C_VEL
LIN {X 0,Y 136.148,Z 723.337,A -85,B 0,C 180,E1 3587.594,E2 3587.594} C_VEL
LIN {X 0,Y 123.255,Z 734.735,A -85,B 0,C 180,E1 3584.849,E2 3584.849} C_VEL
LIN {X 0,Y 110.726,Z 743.904,A -85,B 0,C 180,E1 3581.449,E2 3581.449} C_VEL
LIN {X 0,Y 106.387,Z 746.674,A -85,B 0,C 180,E1 3580.031,E2 3580.031} C_VEL
LIN {X 0,Y 100.145,Z 750.256,A -85,B 0,C 180,E1 3578.403,E2 3578.403} C_VEL
LIN {X 0,Y 86.262,Z 756.396,A -85,B 0,C 180,E1 3575.996,E2 3575.996} C_VEL
LIN {X 0,Y 78.542,Z 759.227,A -85,B 0,C 180,E1 3573.622,E2 3573.622} C_VEL
LIN {X 0,Y 75.948,Z 760.138,A -85,B 0,C 180,E1 3572.23,E2 3572.23} C_VEL
LIN {X 0,Y 62.872,Z 764.131,A -85,B 0,C 180,E1 3561.175,E2 3561.175} C_VEL
LIN {X 0,Y 53.676,Z 766.019,A -85,B 0,C 180,E1 3546.575,E2 3546.575} C_VEL
LIN {X 0,Y 48.85,Z 766.079,A -85,B 0,C 180,E1 3527.866,E2 3527.866} C_VEL
LIN {X 0,Y 48.562,Z 764.748,A -85,B 0,C 180,E1 3511.167,E2 3511.167} C_VEL
LIN {X 0,Y 48.632,Z 762.584,A -85,B 0,C 180,E1 3498.123,E2 3498.123} C_VEL
LIN {X 0,Y 52.117,Z 757.693,A -85,B 0,C 180,E1 3480.065,E2 3480.065} C_VEL
LIN {X 0,Y 58.828,Z 751.676,A -85,B 0,C 180,E1 3467.154,E2 3467.154} C_VEL
LIN {X 0,Y 62.413,Z 748.566,A -85,B 0,C 180,E1 3462.594,E2 3462.594} C_VEL
LIN {X 0,Y 51.174,Z 741.184,A -85,B 0,C 180,E1 3432.278,E2 3432.278} C_VEL
LIN {X 0,Y 51.024,Z 739.137,A -85,B 0,C 180,E1 3423.366,E2 3423.366} C_VEL
LIN {X 0,Y 52.296,Z 736.24,A -85,B 0,C 180,E1 3405.604,E2 3405.604} C_VEL
LIN {X 0,Y 54.257,Z 734.849,A -85,B 0,C 180,E1 3399.5,E2 3399.5} C_VEL
LIN {X 0,Y 57.784,Z 733.261,A -85,B 0,C 180,E1 3389.876,E2 3389.876} C_VEL
LIN {X 0,Y 62.937,Z 731.136,A -85,B 0,C 180,E1 3382.861,E2 3382.861} C_VEL
LIN {X 0,Y 68.894,Z 729.264,A -85,B 0,C 180,E1 3375.839,E2 3375.839} C_VEL
LIN {X 0,Y 76.377,Z 726.496,A -85,B 0,C 180,E1 3370.594,E2 3370.594} C_VEL
LIN {X 0,Y 83.252,Z 724.561,A -85,B 0,C 180,E1 3366.155,E2 3366.155} C_VEL
LIN {X 0,Y 73.644,Z 734.549,A -85,B 0,C 180,E1 3360.165,E2 3360.165} C_VEL
LIN {X 0,Y 63.709,Z 743.748,A -85,B 0,C 180,E1 3351.17,E2 3351.17} C_VEL
LIN {X 0,Y 55.65,Z 750.771,A -85,B 0,C 180,E1 3339.317,E2 3339.317} C_VEL
LIN {X 0,Y 50.071,Z 756.343,A -85,B 0,C 180,E1 3323.131,E2 3323.131} C_VEL
LIN {X 0,Y 48.394,Z 759.667,A -85,B 0,C 180,E1 3306.901,E2 3306.901} C_VEL
LIN {X 0,Y 49.771,Z 761.695,A -85,B 0,C 180,E1 3289.771,E2 3289.771} C_VEL
LIN {X 0,Y 55.608,Z 762.328,A -85,B 0,C 180,E1 3272.341,E2 3272.341} C_VEL
LIN {X 0,Y 64.715,Z 761.262,A -85,B 0,C 180,E1 3259.562,E2 3259.562} C_VEL
LIN {X 0,Y 77.063,Z 758.174,A -85,B 0,C 180,E1 3249.631,E2 3249.631} C_VEL
LIN {X 0,Y 90.096,Z 753.471,A -85,B 0,C 180,E1 3242.969,E2 3242.969} C_VEL
LIN {X 0,Y 104.034,Z 746.718,A -85,B 0,C 180,E1 3238.035,E2 3238.035} C_VEL
LIN {X 0,Y 117.126,Z 738.685,A -85,B 0,C 180,E1 3234.614,E2 3234.614} C_VEL
LIN {X 0,Y 129.766,Z 728.943,A -85,B 0,C 180,E1 3232.029,E2 3232.029} C_VEL
LIN {X 0,Y 135.48,Z 723.816,A -85,B 0,C 180,E1 3231.032,E2 3231.032} C_VEL
LIN {X 0,Y 122.347,Z 734.863,A -85,B 0,C 180,E1 3228.689,E2 3228.689} C_VEL
LIN {X 0,Y 109.158,Z 744.014,A -85,B 0,C 180,E1 3225.683,E2 3225.683} C_VEL
LIN {X 0,Y 94.094,Z 752.431,A -85,B 0,C 180,E1 3221.015,E2 3221.015} C_VEL
LIN {X 0,Y 80.557,Z 758.406,A -85,B 0,C 180,E1 3214.947,E2 3214.947} C_VEL
LIN {X 0,Y 75.948,Z 760.138,A -85,B 0,C 180,E1 3212.23,E2 3212.23} C_VEL
LIN {X 0,Y 69.714,Z 762.031,A -85,B 0,C 180,E1 3208.877,E2 3208.877} C_VEL
LIN {X 0,Y 57.573,Z 764.468,A -85,B 0,C 180,E1 3202.971,E2 3202.971} C_VEL
LIN {X 0,Y 49.743,Z 765.445,A -85,B 0,C 180,E1 3196.333,E2 3196.333} C_VEL
LIN {X 0,Y 47.443,Z 765.646,A -85,B 0,C 180,E1 3192.643,E2 3192.643} C_VEL
LIN {X 0,Y 41.198,Z 765.581,A -85,B 0,C 180,E1 3171.332,E2 3171.332} C_VEL
LIN {X 0,Y 40.571,Z 764.124,A -85,B 0,C 180,E1 3151.397,E2 3151.397} C_VEL
LIN {X 0,Y 40.775,Z 761.817,A -85,B 0,C 180,E1 3135.79,E2 3135.79} C_VEL
LIN {X 0,Y 45.292,Z 756.771,A -85,B 0,C 180,E1 3114.956,E2 3114.956} C_VEL
LIN {X 0,Y 52.788,Z 750.756,A -85,B 0,C 180,E1 3101.519,E2 3101.519} C_VEL
LIN {X 0,Y 44.063,Z 744.166,A -85,B 0,C 180,E1 3067.82,E2 3067.82} C_VEL
LIN {X 0,Y 44.072,Z 743.062,A -85,B 0,C 180,E1 3061.295,E2 3061.295} C_VEL
LIN {X 0,Y 46.096,Z 740.44,A -85,B 0,C 180,E1 3042.317,E2 3042.317} C_VEL
LIN {X 0,Y 48.366,Z 739.221,A -85,B 0,C 180,E1 3035.573,E2 3035.573} C_VEL
LIN {X 0,Y 53.297,Z 737.436,A -85,B 0,C 180,E1 3024.434,E2 3024.434} C_VEL
LIN {X 0,Y 58.435,Z 735.657,A -85,B 0,C 180,E1 3018.135,E2 3018.135} C_VEL
LIN {X 0,Y 65.906,Z 733.598,A -85,B 0,C 180,E1 3010.659,E2 3010.659} C_VEL
LIN {X 0,Y 71.597,Z 731.764,A -85,B 0,C 180,E1 3007.045,E2 3007.045} C_VEL
LIN {X 0,Y 61.08,Z 741.123,A -85,B 0,C 180,E1 2999.423,E2 2999.423} C_VEL
LIN {X 0,Y 51.351,Z 748.855,A -85,B 0,C 180,E1 2988.164,E2 2988.164} C_VEL
LIN {X 0,Y 44.033,Z 754.84,A -85,B 0,C 180,E1 2972.3,E2 2972.3} C_VEL
LIN {X 0,Y 40.624,Z 758.925,A -85,B 0,C 180,E1 2952.838,E2 2952.838} C_VEL
LIN {X 0,Y 41.171,Z 761.455,A -85,B 0,C 180,E1 2932.637,E2 2932.637} C_VEL
LIN {X 0,Y 46.909,Z 762.746,A -85,B 0,C 180,E1 2911.533,E2 2911.533} C_VEL
LIN {X 0,Y 56.45,Z 762.234,A -85,B 0,C 180,E1 2897.008,E2 2897.008} C_VEL
LIN {X 0,Y 69.416,Z 759.848,A -85,B 0,C 180,E1 2886.436,E2 2886.436} C_VEL
LIN {X 0,Y 82.977,Z 755.82,A -85,B 0,C 180,E1 2879.718,E2 2879.718} C_VEL
LIN {X 0,Y 98.076,Z 749.511,A -85,B 0,C 180,E1 2874.738,E2 2874.738} C_VEL
LIN {X 0,Y 111.158,Z 742.379,A -85,B 0,C 180,E1 2871.624,E2 2871.624} C_VEL
LIN {X 0,Y 113.601,Z 740.829,A -85,B 0,C 180,E1 2871.063,E2 2871.063} C_VEL
LIN {X 0,Y 99.18,Z 749.152,A -85,B 0,C 180,E1 2867.894,E2 2867.894} C_VEL
LIN {X 0,Y 84.518,Z 755.857,A -85,B 0,C 180,E1 2863.355,E2 2863.355} C_VEL
LIN {X 0,Y 69.548,Z 761.078,A -85,B 0,C 180,E1 2856.266,E2 2856.266} C_VEL
LIN {X 0,Y 56.658,Z 764.252,A -85,B 0,C 180,E1 2846.019,E2 2846.019} C_VEL
LIN {X 0,Y 47.443,Z 765.646,A -85,B 0,C 180,E1 2832.643,E2 2832.643} C_VEL
LIN {X 0,Y 42.964,Z 765.79,A -85,B 0,C 180,E1 2823.71,E2 2823.71} C_VEL
LIN {X 0,Y 37.081,Z 765.186,A -85,B 0,C 180,E1 2810.042,E2 2810.042} C_VEL
LIN {X 0,Y 32.516,Z 762.639,A -85,B 0,C 180,E1 2784.104,E2 2784.104} C_VEL
LIN {X 0,Y 35.198,Z 758.703,A -85,B 0,C 180,E1 2759.228,E2 2759.228} C_VEL
LIN {X 0,Y 43.194,Z 752.736,A -85,B 0,C 180,E1 2740.005,E2 2740.005} C_VEL
LIN {X 0,Y 37.08,Z 746.957,A -85,B 0,C 180,E1 2701.54,E2 2701.54} C_VEL
LIN {X 0,Y 39.91,Z 744.302,A -85,B 0,C 180,E1 2677.921,E2 2677.921} C_VEL
LIN {X 0,Y 42.198,Z 743.321,A -85,B 0,C 180,E1 2671.707,E2 2671.707} C_VEL
LIN {X 0,Y 48.564,Z 741.49,A -85,B 0,C 180,E1 2658.783,E2 2658.783} C_VEL
LIN {X 0,Y 54.255,Z 739.826,A -85,B 0,C 180,E1 2652.504,E2 2652.504} C_VEL
LIN {X 0,Y 59.048,Z 738.776,A -85,B 0,C 180,E1 2647.726,E2 2647.726} C_VEL
LIN {X 0,Y 47.701,Z 747.243,A -85,B 0,C 180,E1 2637.475,E2 2637.475} C_VEL
LIN {X 0,Y 38.542,Z 753.625,A -85,B 0,C 180,E1 2621.994,E2 2621.994} C_VEL
LIN {X 0,Y 32.962,Z 758.553,A -85,B 0,C 180,E1 2597.76,E2 2597.76} C_VEL
LIN {X 0,Y 33.031,Z 761.417,A -85,B 0,C 180,E1 2572.767,E2 2572.767} C_VEL
LIN {X 0,Y 38.807,Z 762.993,A -85,B 0,C 180,E1 2548.869,E2 2548.869} C_VEL
LIN {X 0,Y 50.305,Z 762.877,A -85,B 0,C 180,E1 2531.469,E2 2531.469} C_VEL
LIN {X 0,Y 63.997,Z 760.922,A -85,B 0,C 180,E1 2521.333,E2 2521.333} C_VEL
LIN {X 0,Y 79.309,Z 756.962,A -85,B 0,C 180,E1 2514.754,E2 2514.754} C_VEL
LIN {X 0,Y 91.563,Z 752.466,A -85,B 0,C 180,E1 2511.16,E2 2511.16} C_VEL
LIN {X 0,Y 75.117,Z 758.616,A -85,B 0,C 180,E1 2506.293,E2 2506.293} C_VEL
LIN {X 0,Y 59.971,Z 762.654,A -85,B 0,C 180,E1 2498.981,E2 2498.981} C_VEL
LIN {X 0,Y 45.721,Z 764.96,A -85,B 0,C 180,E1 2486.178,E2 2486.178} C_VEL
LIN {X 0,Y 35.845,Z 765.359,A -85,B 0,C 180,E1 2465.835,E2 2465.835} C_VEL
LIN {X 0,Y 32.426,Z 764.054,A -85,B 0,C 180,E1 2438.849,E2 2438.849} C_VEL
LIN {X 0,Y 32.576,Z 763.11,A -85,B 0,C 180,E1 2428.222,E2 2428.222} C_VEL
LIN {X 0,Y 32.516,Z 762.639,A -85,B 0,C 180,E1 2424.104,E2 2424.104} C_VEL
LIN {X 0,Y 31.778,Z 761.477,A -85,B 0,C 180,E1 2415.116,E2 2415.116} C_VEL
LIN {X 0,Y 29.954,Z 757.42,A -85,B 0,C 180,E1 2389.263,E2 2389.263} C_VEL
LIN {X 0,Y 31.735,Z 755.808,A -85,B 0,C 180,E1 2382.162,E2 2382.162} C_VEL
LIN {X 0,Y 33.735,Z 754.554,A -85,B 0,C 180,E1 2377.999,E2 2377.999} C_VEL
LIN {X 0,Y 29.833,Z 750.319,A -85,B 0,C 180,E1 2339.993,E2 2339.993} C_VEL
LIN {X 0,Y 33.883,Z 747.818,A -85,B 0,C 180,E1 2311.819,E2 2311.819} C_VEL
LIN {X 0,Y 36.59,Z 746.95,A -85,B 0,C 180,E1 2304.974,E2 2304.974} C_VEL
LIN {X 0,Y 45.04,Z 745.008,A -85,B 0,C 180,E1 2290.987,E2 2290.987} C_VEL
LIN {X 0,Y 46.78,Z 744.592,A -85,B 0,C 180,E1 2289.106,E2 2289.106} C_VEL
LIN {X 0,Y 35.742,Z 751.501,A -85,B 0,C 180,E1 2276.608,E2 2276.608} C_VEL
LIN {X 0,Y 26.735,Z 757.193,A -85,B 0,C 180,E1 2252.167,E2 2252.167} C_VEL
LIN {X 0,Y 24.458,Z 760.653,A -85,B 0,C 180,E1 2220.652,E2 2220.652} C_VEL
LIN {X 0,Y 29.577,Z 762.918,A -85,B 0,C 180,E1 2188.255,E2 2188.255} C_VEL
LIN {X 0,Y 41.36,Z 763.573,A -85,B 0,C 180,E1 2167.744,E2 2167.744} C_VEL
LIN {X 0,Y 55.037,Z 762.536,A -85,B 0,C 180,E1 2157.403,E2 2157.403} C_VEL
LIN {X 0,Y 69.552,Z 759.824,A -85,B 0,C 180,E1 2151.325,E2 2151.325} C_VEL
LIN {X 0,Y 53.884,Z 763.191,A -85,B 0,C 180,E1 2144.729,E2 2144.729} C_VEL
LIN {X 0,Y 38.52,Z 764.842,A -85,B 0,C 180,E1 2131.915,E2 2131.915} C_VEL
LIN {X 0,Y 27.583,Z 764.667,A -85,B 0,C 180,E1 2108.013,E2 2108.013} C_VEL
LIN {X 0,Y 24.516,Z 762.987,A -85,B 0,C 180,E1 2074.653,E2 2074.653} C_VEL
LIN {X 0,Y 24.53,Z 762.012,A -85,B 0,C 180,E1 2062.951,E2 2062.951} C_VEL
LIN {X 0,Y 28.553,Z 757.803,A -85,B 0,C 180,E1 2030.9,E2 2030.9} C_VEL
LIN {X 0,Y 31.735,Z 755.808,A -85,B 0,C 180,E1 2022.162,E2 2022.162} C_VEL
LIN {X 0,Y 32.189,Z 754.973,A -85,B 0,C 180,E1 2018.325,E2 2018.325} C_VEL
LIN {X 0,Y 31.169,Z 754.229,A -85,B 0,C 180,E1 2012.919,E2 2012.919} C_VEL
LIN {X 0,Y 28.418,Z 753.723,A -85,B 0,C 180,E1 2004.855,E2 2004.855} C_VEL
LIN {X 0,Y 22.653,Z 753.395,A -85,B 0,C 180,E1 1980.587,E2 1980.587} C_VEL
LIN {X 0,Y 22.534,Z 753.135,A -85,B 0,C 180,E1 1973.574,E2 1973.574} C_VEL
LIN {X 0,Y 29.617,Z 750.619,A -85,B 0,C 180,E1 1940.092,E2 1940.092} C_VEL
LIN {X 0,Y 33.916,Z 749.822,A -85,B 0,C 180,E1 1931.015,E2 1931.015} C_VEL
LIN {X 0,Y 22.242,Z 755.859,A -85,B 0,C 180,E1 1911.107,E2 1911.107} C_VEL
LIN {X 0,Y 16.487,Z 759.847,A -85,B 0,C 180,E1 1872.389,E2 1872.389} C_VEL
LIN {X 0,Y 20.242,Z 762.521,A -85,B 0,C 180,E1 1827.309,E2 1827.309} C_VEL
LIN {X 0,Y 32.997,Z 763.94,A -85,B 0,C 180,E1 1801.631,E2 1801.631} C_VEL
LIN {X 0,Y 47.514,Z 763.62,A -85,B 0,C 180,E1 1791.415,E2 1791.415} C_VEL
LIN {X 0,Y 31.019,Z 764.535,A -85,B 0,C 180,E1 1779.133,E2 1779.133} C_VEL
LIN {X 0,Y 18.891,Z 763.659,A -85,B 0,C 180,E1 1749.386,E2 1749.386} C_VEL
LIN {X 0,Y 16.629,Z 761.89,A -85,B 0,C 180,E1 1709.963,E2 1709.963} C_VEL
LIN {X 0,Y 20.9,Z 757.891,A -85,B 0,C 180,E1 1664.1,E2 1664.1} C_VEL
LIN {X 0,Y 24.287,Z 756.124,A -85,B 0,C 180,E1 1654.532,E2 1654.532} C_VEL
LIN {X 0,Y 22.456,Z 753.317,A -85,B 0,C 180,E1 1617.439,E2 1617.439} C_VEL
LIN {X 0,Y 22.534,Z 753.135,A -85,B 0,C 180,E1 1613.574,E2 1613.574} C_VEL
LIN {X 0,Y 22.022,Z 753.175,A -85,B 0,C 180,E1 1606.683,E2 1606.683} C_VEL
LIN {X 0,Y 20.063,Z 753.934,A -85,B 0,C 180,E1 1597.921,E2 1597.921} C_VEL
LIN {X 0,Y 16.567,Z 755.444,A -85,B 0,C 180,E1 1586.19,E2 1586.19} C_VEL
LIN {X 0,Y 12.133,Z 757.333,A -85,B 0,C 180,E1 1569.329,E2 1569.329} C_VEL
LIN {X 0,Y 7.838,Z 759.988,A -85,B 0,C 180,E1 1516.276,E2 1516.276} C_VEL
LIN {X 0,Y 11.235,Z 761.902,A -85,B 0,C 180,E1 1462.18,E2 1462.18} C_VEL
LIN {X 0,Y 25.265,Z 763.997,A -85,B 0,C 180,E1 1431.46,E2 1431.46} C_VEL
LIN {X 0,Y 10.805,Z 762.502,A -85,B 0,C 180,E1 1397.668,E2 1397.668} C_VEL
LIN {X 0,Y 8.617,Z 761.164,A -85,B 0,C 180,E1 1349.928,E2 1349.928} C_VEL
LIN {X 0,Y 15.028,Z 757.449,A -85,B 0,C 180,E1 1286.14,E2 1286.14} C_VEL
LIN {X 0,Y 15.112,Z 755.87,A -85,B 0,C 180,E1 1249.853,E2 1249.853} C_VEL
LIN {X 0,Y 20.854,Z 754.362,A -85,B 0,C 180,E1 1215.308,E2 1215.308} C_VEL
LIN {X 0,Y 9.615,Z 759.087,A -85,B 0,C 180,E1 1176.034,E2 1176.034} C_VEL
LIN {X 0,Y 11.235,Z 761.902,A -85,B 0,C 180,E1 1102.18,E2 1102.18} C_VEL
LIN {X 0,Y 10.709,Z 762.006,A -85,B 0,C 180,E1 1095.717,E2 1095.717} C_VEL
LIN {X 0,Y 8,Z 761.808,A -85,B 0,C 180,E1 1087.278,E2 1087.278} C_VEL
LIN {X 0,Y 3.029,Z 761.038,A -85,B 0,C 180,E1 1073.274,E2 1073.274} C_VEL
LIN {X 0,Y 0.837,Z 760.527,A -85,B 0,C 180,E1 1082.641,E2 1082.641} C_VEL
LIN {X 0,Y 7.884,Z 758.174,A -85,B 0,C 180,E1 1236.325,E2 1236.325} C_VEL
LIN {X 0,Y 6.733,Z 758.631,A -85,B 0,C 180,E1 1257.123,E2 1257.123} C_VEL
LIN {X 0,Y 1.096,Z 760.611,A -85,B 0,C 180,E1 1414.419,E2 1414.419} C_VEL
LIN {X 0,Y 1.485,Z 760.689,A -85,B 0,C 180,E1 1430.199,E2 1430.199} C_VEL
LIN {X 0,Y 0.837,Z 760.527,A -85,B 0,C 180,E1 1442.641,E2 1442.641} C_VEL
LIN {X 0,Y 1.794,Z 762.465,A -85,B 0,C 180,E1 1583.024,E2 1583.024} C_VEL
LIN {X 0,Y 1.794,Z 799,A -85,B 0,C 180,E1 1583.024,E2 1583.024} C_VEL
LIN {X 0,Y 1.794,Z 799,A -85,B 0,C 180,E1 1583.024,E2 1583.024}

QRS_NEXT_CUT()

QRS_NEXT()
QRS_HOME()

END
